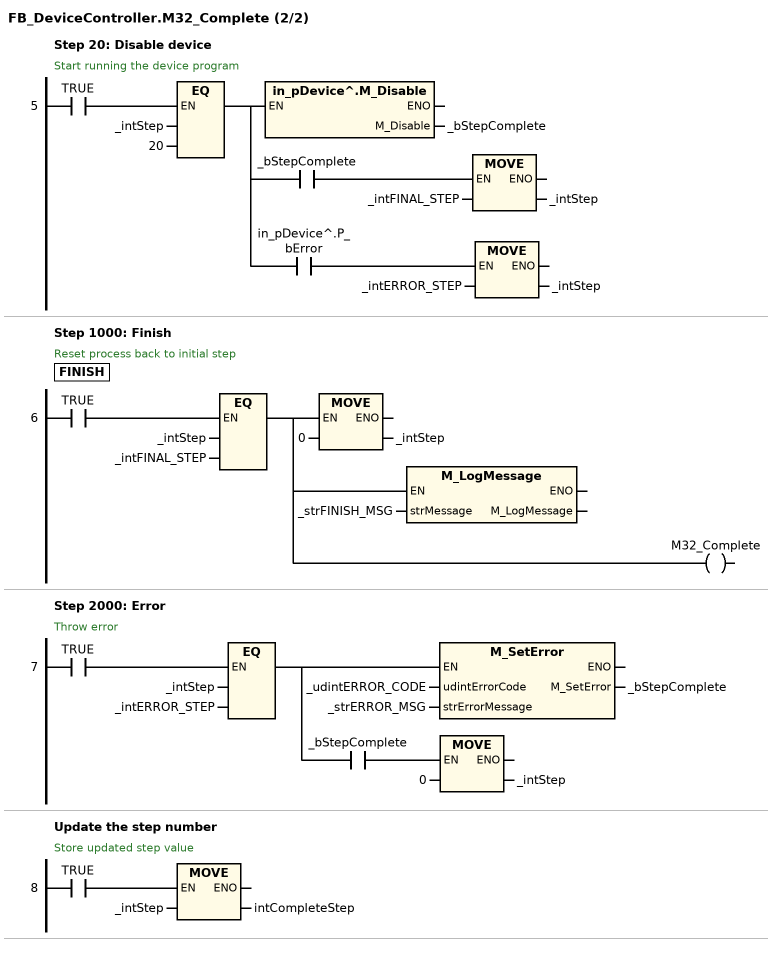
// NETWORK 5: Step 20: Disable device
// Start running the device program
_w6 := _intStep = 20;
IF _w6 THEN _bStepComplete := in_pDevice^.M_Disable(); END_IF
IF _w6 AND _bStepComplete THEN _intStep := _intFINAL_STEP; END_IF
IF _w6 AND in_pDevice^.P_bError THEN _intStep := _intERROR_STEP; END_IF

// NETWORK 6: Step 1000: Finish
// Reset process back to initial step
FINISH:
_w7 := _intStep = _intFINAL_STEP;
IF _w7 THEN _intStep := 0; END_IF
IF _w7 THEN M_LogMessage(strMessage := _strFINISH_MSG); END_IF
M32_Complete := _w7;

// NETWORK 7: Step 2000: Error
// Throw error
_w8 := _intStep = _intERROR_STEP;
IF _w8 THEN
    _bStepComplete := M_SetError(udintErrorCode := _udintERROR_CODE, strErrorMessage := _strERROR_MSG);
END_IF
IF _w8 AND _bStepComplete THEN _intStep := 0; END_IF

// NETWORK 8: Update the step number
// Store updated step value
intCompleteStep := _intStep;
END_METHOD

(* Pauses the device then returns TRUE. *)
METHOD M40_Hold : BOOL
VAR CONSTANT
	_udintERROR_CODE: UDINT := E_DeviceControllerError.HoldError;
	_strERROR_MSG: T_MaxString := 'Error while trying to hold device!';
	_intFINAL_STEP : INT := 1000;
	_intERROR_STEP : INT := 2000;
	_strSTART_MSG: T_MaxString := 'Holding device';
	_strFINISH_MSG: T_MaxString := 'Device held';
END_VAR
VAR
	_bStepComplete: BOOL;
	_intStep: INT;
END_VAR
VAR_INST // added by the converter: edge detectors and wires of the graphical bodies
    _w1, _w2, _w3, _w4, _w5, _w6, _w7 : BOOL;
END_VAR
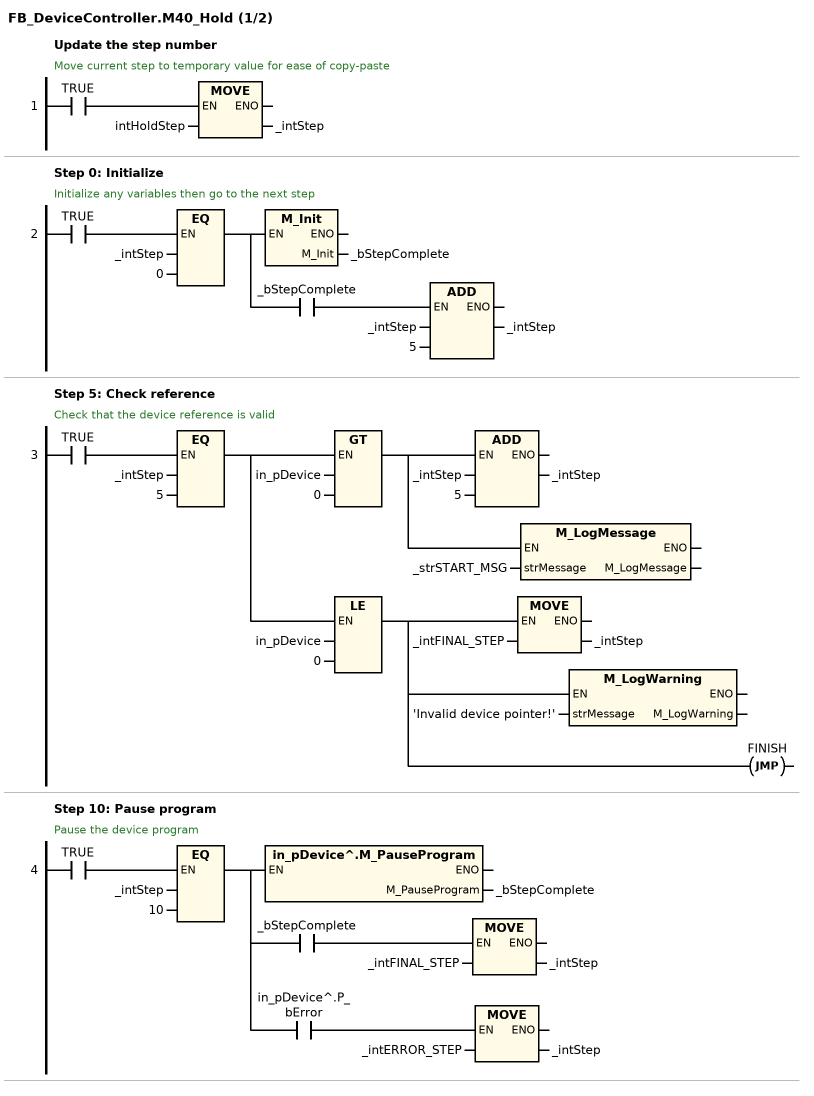
// NETWORK 1: Update the step number
// Move current step to temporary value for ease of copy-paste
_intStep := intHoldStep;

// NETWORK 2: Step 0: Initialize
// Initialize any variables then go to the next step
_w1 := _intStep = 0;
IF _w1 THEN _bStepComplete := M_Init(); END_IF
IF _w1 AND _bStepComplete THEN _intStep := _intStep + 5; END_IF

// NETWORK 3: Step 5: Check reference
// Check that the device reference is valid
_w2 := _intStep = 5;
_w3 := _w2 AND in_pDevice > 0;
IF _w3 THEN _intStep := _intStep + 5; END_IF
IF _w3 THEN M_LogMessage(strMessage := _strSTART_MSG); END_IF
_w4 := _w2 AND in_pDevice <= 0;
IF _w4 THEN _intStep := _intFINAL_STEP; END_IF
IF _w4 THEN M_LogWarning(strMessage := 'Invalid device pointer!'); END_IF
IF _w4 THEN JMP FINISH; END_IF

// NETWORK 4: Step 10: Pause program
// Pause the device program
_w5 := _intStep = 10;
IF _w5 THEN _bStepComplete := in_pDevice^.M_PauseProgram(); END_IF
IF _w5 AND _bStepComplete THEN _intStep := _intFINAL_STEP; END_IF
IF _w5 AND in_pDevice^.P_bError THEN _intStep := _intERROR_STEP; END_IF

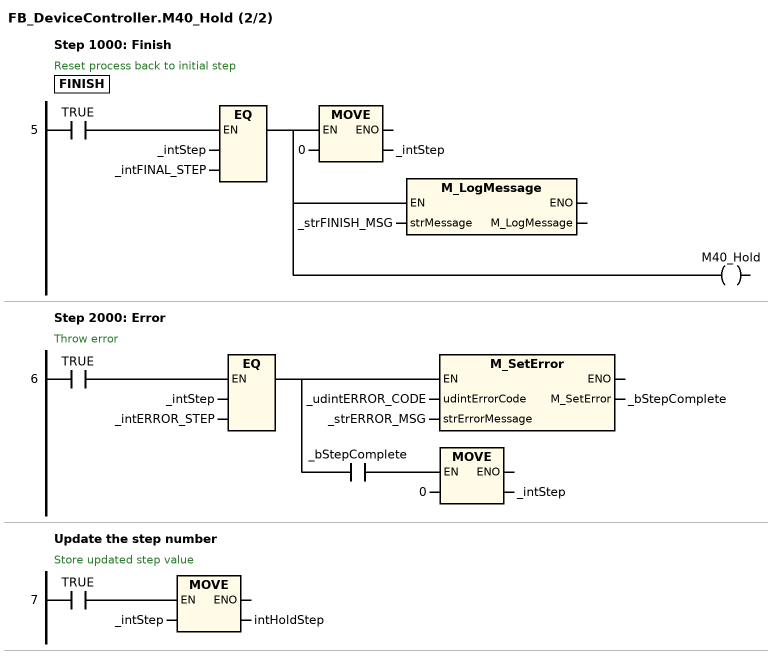
// NETWORK 5: Step 1000: Finish
// Reset process back to initial step
FINISH:
_w6 := _intStep = _intFINAL_STEP;
IF _w6 THEN _intStep := 0; END_IF
IF _w6 THEN M_LogMessage(strMessage := _strFINISH_MSG); END_IF
M40_Hold := _w6;

// NETWORK 6: Step 2000: Error
// Throw error
_w7 := _intStep = _intERROR_STEP;
IF _w7 THEN
    _bStepComplete := M_SetError(udintErrorCode := _udintERROR_CODE, strErrorMessage := _strERROR_MSG);
END_IF
IF _w7 AND _bStepComplete THEN _intStep := 0; END_IF

// NETWORK 7: Update the step number
// Store updated step value
intHoldStep := _intStep;
END_METHOD

(* Unpauses the device then returns TRUE. *)
METHOD M42_Unhold : BOOL
VAR CONSTANT
	_udintERROR_CODE: UDINT := E_DeviceControllerError.UnholdError;
	_strERROR_MSG: T_MaxString := 'Error while trying to unhold device!';
	_intFINAL_STEP : INT := 1000;
	_intERROR_STEP : INT := 2000;
	_strSTART_MSG: T_MaxString := 'Unholding device';
	_strFINISH_MSG: T_MaxString := 'Device unheld';
END_VAR
VAR
	_bStepComplete: BOOL;
	_intStep: INT;
END_VAR
VAR_INST // added by the converter: edge detectors and wires of the graphical bodies
    _w1, _w2, _w3, _w4, _w5, _w6, _w7 : BOOL;
END_VAR
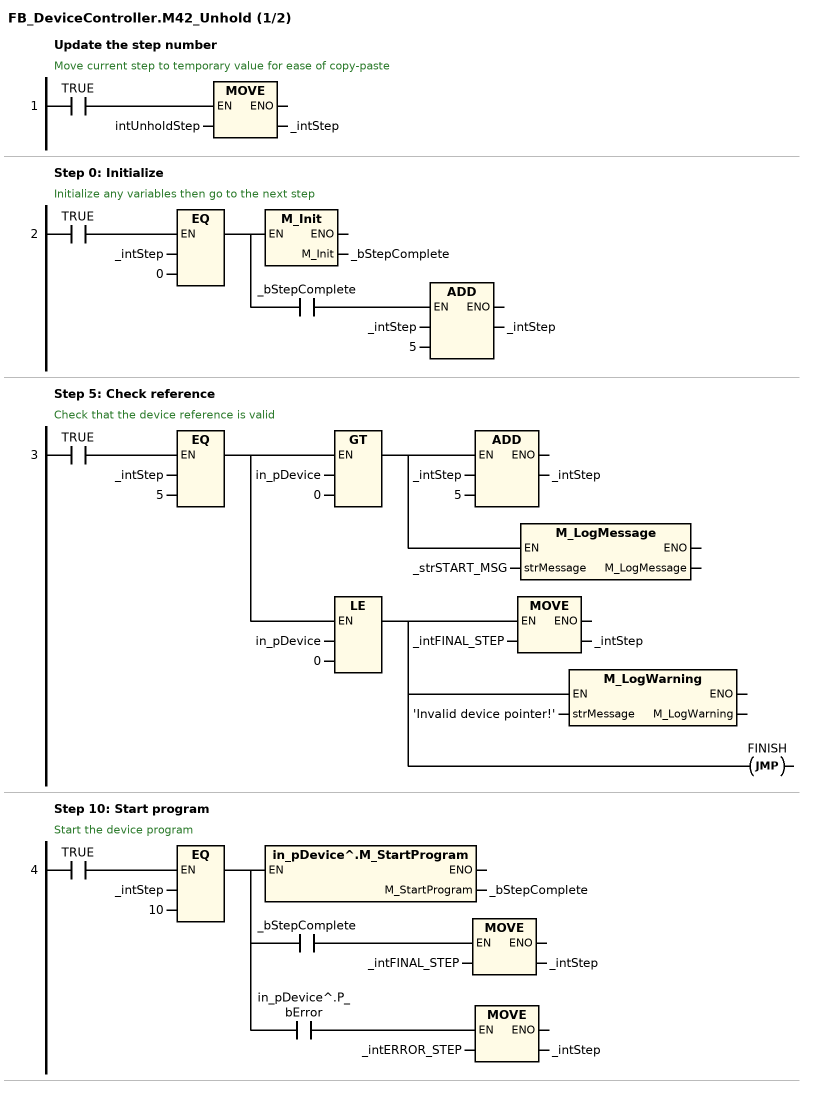
// NETWORK 1: Update the step number
// Move current step to temporary value for ease of copy-paste
_intStep := intUnholdStep;

// NETWORK 2: Step 0: Initialize
// Initialize any variables then go to the next step
_w1 := _intStep = 0;
IF _w1 THEN _bStepComplete := M_Init(); END_IF
IF _w1 AND _bStepComplete THEN _intStep := _intStep + 5; END_IF

// NETWORK 3: Step 5: Check reference
// Check that the device reference is valid
_w2 := _intStep = 5;
_w3 := _w2 AND in_pDevice > 0;
IF _w3 THEN _intStep := _intStep + 5; END_IF
IF _w3 THEN M_LogMessage(strMessage := _strSTART_MSG); END_IF
_w4 := _w2 AND in_pDevice <= 0;
IF _w4 THEN _intStep := _intFINAL_STEP; END_IF
IF _w4 THEN M_LogWarning(strMessage := 'Invalid device pointer!'); END_IF
IF _w4 THEN JMP FINISH; END_IF

// NETWORK 4: Step 10: Start program
// Start the device program
_w5 := _intStep = 10;
IF _w5 THEN _bStepComplete := in_pDevice^.M_StartProgram(); END_IF
IF _w5 AND _bStepComplete THEN _intStep := _intFINAL_STEP; END_IF
IF _w5 AND in_pDevice^.P_bError THEN _intStep := _intERROR_STEP; END_IF

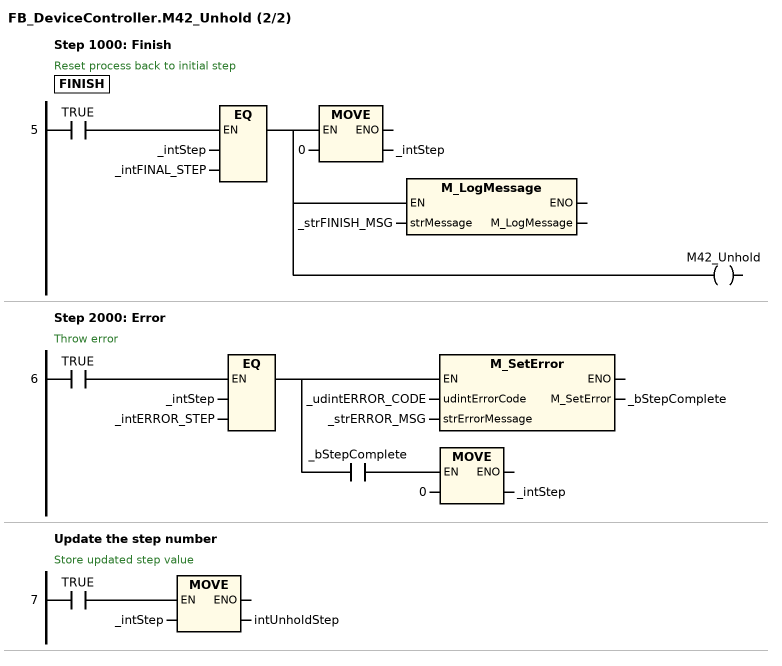
// NETWORK 5: Step 1000: Finish
// Reset process back to initial step
FINISH:
_w6 := _intStep = _intFINAL_STEP;
IF _w6 THEN _intStep := 0; END_IF
IF _w6 THEN M_LogMessage(strMessage := _strFINISH_MSG); END_IF
M42_Unhold := _w6;

// NETWORK 6: Step 2000: Error
// Throw error
_w7 := _intStep = _intERROR_STEP;
IF _w7 THEN
    _bStepComplete := M_SetError(udintErrorCode := _udintERROR_CODE, strErrorMessage := _strERROR_MSG);
END_IF
IF _w7 AND _bStepComplete THEN _intStep := 0; END_IF

// NETWORK 7: Update the step number
// Store updated step value
intUnholdStep := _intStep;
END_METHOD

(* Pauses the device then returns TRUE. *)
METHOD M50_Suspend : BOOL
VAR CONSTANT
	_udintERROR_CODE: UDINT := E_DeviceControllerError.SuspendError;
	_strERROR_MSG: T_MaxString := 'Error while trying to suspend device!';
	_intFINAL_STEP : INT := 1000;
	_intERROR_STEP : INT := 2000;
	_strSTART_MSG: T_MaxString := 'Suspending device';
	_strFINISH_MSG: T_MaxString := 'Device suspended';
END_VAR
VAR
	_bStepComplete: BOOL;
	_intStep: INT;
END_VAR
VAR_INST // added by the converter: edge detectors and wires of the graphical bodies
    _w1, _w2, _w3, _w4, _w5, _w6, _w7 : BOOL;
END_VAR
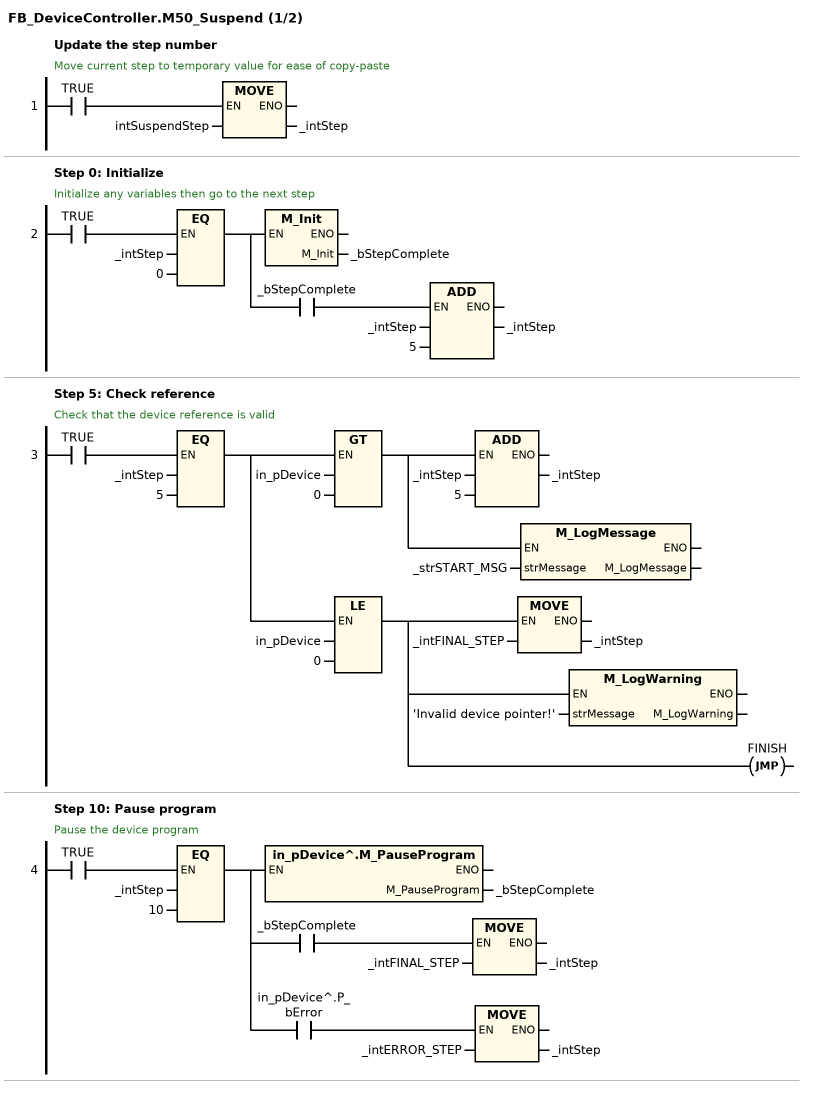
// NETWORK 1: Update the step number
// Move current step to temporary value for ease of copy-paste
_intStep := intSuspendStep;

// NETWORK 2: Step 0: Initialize
// Initialize any variables then go to the next step
_w1 := _intStep = 0;
IF _w1 THEN _bStepComplete := M_Init(); END_IF
IF _w1 AND _bStepComplete THEN _intStep := _intStep + 5; END_IF

// NETWORK 3: Step 5: Check reference
// Check that the device reference is valid
_w2 := _intStep = 5;
_w3 := _w2 AND in_pDevice > 0;
IF _w3 THEN _intStep := _intStep + 5; END_IF
IF _w3 THEN M_LogMessage(strMessage := _strSTART_MSG); END_IF
_w4 := _w2 AND in_pDevice <= 0;
IF _w4 THEN _intStep := _intFINAL_STEP; END_IF
IF _w4 THEN M_LogWarning(strMessage := 'Invalid device pointer!'); END_IF
IF _w4 THEN JMP FINISH; END_IF

// NETWORK 4: Step 10: Pause program
// Pause the device program
_w5 := _intStep = 10;
IF _w5 THEN _bStepComplete := in_pDevice^.M_PauseProgram(); END_IF
IF _w5 AND _bStepComplete THEN _intStep := _intFINAL_STEP; END_IF
IF _w5 AND in_pDevice^.P_bError THEN _intStep := _intERROR_STEP; END_IF

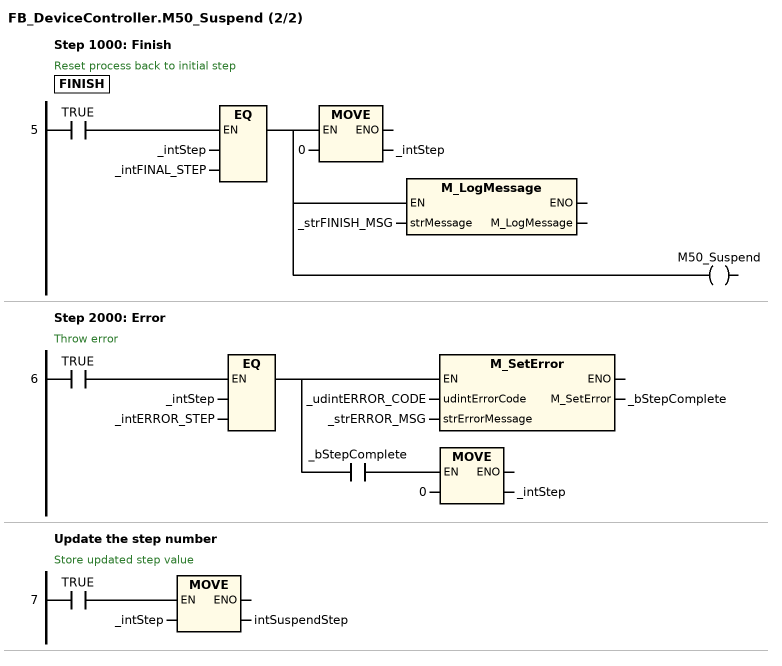
// NETWORK 5: Step 1000: Finish
// Reset process back to initial step
FINISH:
_w6 := _intStep = _intFINAL_STEP;
IF _w6 THEN _intStep := 0; END_IF
IF _w6 THEN M_LogMessage(strMessage := _strFINISH_MSG); END_IF
M50_Suspend := _w6;

// NETWORK 6: Step 2000: Error
// Throw error
_w7 := _intStep = _intERROR_STEP;
IF _w7 THEN
    _bStepComplete := M_SetError(udintErrorCode := _udintERROR_CODE, strErrorMessage := _strERROR_MSG);
END_IF
IF _w7 AND _bStepComplete THEN _intStep := 0; END_IF

// NETWORK 7: Update the step number
// Store updated step value
intSuspendStep := _intStep;
END_METHOD

(* Unpauses the device then returns TRUE. *)
METHOD M52_Unsuspend : BOOL
VAR CONSTANT
	_udintERROR_CODE: UDINT := E_DeviceControllerError.ResetError;
	_strERROR_MSG: T_MaxString := 'Error while trying to reset device!';
	_intFINAL_STEP : INT := 1000;
	_intERROR_STEP : INT := 2000;
	_strSTART_MSG: T_MaxString := 'Unsuspending device';
	_strFINISH_MSG: T_MaxString := 'Device unsuspended';
END_VAR
VAR
	_bStepComplete: BOOL;
	_intStep: INT;
END_VAR
VAR_INST // added by the converter: edge detectors and wires of the graphical bodies
    _w1, _w2, _w3, _w4, _w5, _w6, _w7 : BOOL;
END_VAR
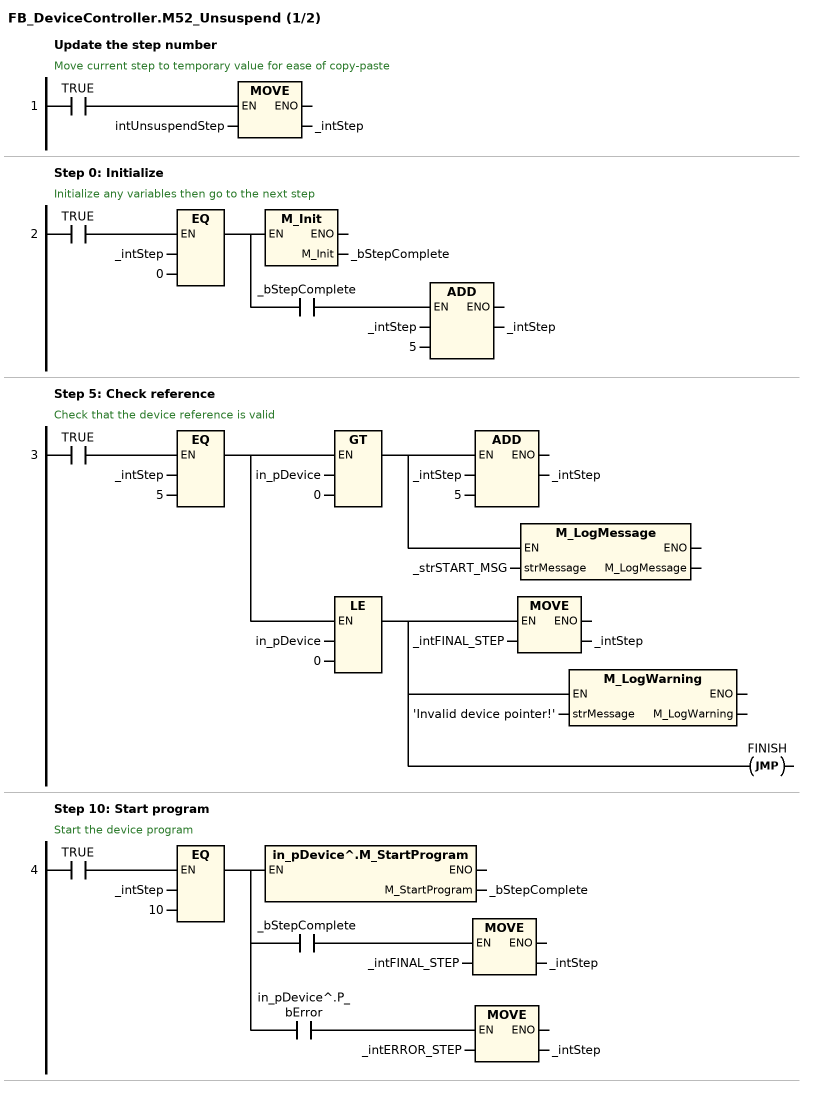
// NETWORK 1: Update the step number
// Move current step to temporary value for ease of copy-paste
_intStep := intUnsuspendStep;

// NETWORK 2: Step 0: Initialize
// Initialize any variables then go to the next step
_w1 := _intStep = 0;
IF _w1 THEN _bStepComplete := M_Init(); END_IF
IF _w1 AND _bStepComplete THEN _intStep := _intStep + 5; END_IF

// NETWORK 3: Step 5: Check reference
// Check that the device reference is valid
_w2 := _intStep = 5;
_w3 := _w2 AND in_pDevice > 0;
IF _w3 THEN _intStep := _intStep + 5; END_IF
IF _w3 THEN M_LogMessage(strMessage := _strSTART_MSG); END_IF
_w4 := _w2 AND in_pDevice <= 0;
IF _w4 THEN _intStep := _intFINAL_STEP; END_IF
IF _w4 THEN M_LogWarning(strMessage := 'Invalid device pointer!'); END_IF
IF _w4 THEN JMP FINISH; END_IF

// NETWORK 4: Step 10: Start program
// Start the device program
_w5 := _intStep = 10;
IF _w5 THEN _bStepComplete := in_pDevice^.M_StartProgram(); END_IF
IF _w5 AND _bStepComplete THEN _intStep := _intFINAL_STEP; END_IF
IF _w5 AND in_pDevice^.P_bError THEN _intStep := _intERROR_STEP; END_IF

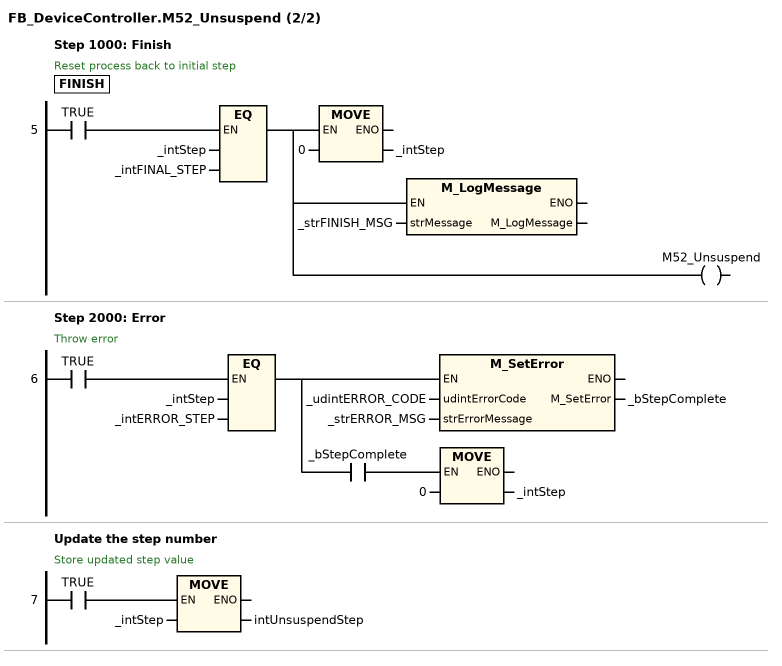
// NETWORK 5: Step 1000: Finish
// Reset process back to initial step
FINISH:
_w6 := _intStep = _intFINAL_STEP;
IF _w6 THEN _intStep := 0; END_IF
IF _w6 THEN M_LogMessage(strMessage := _strFINISH_MSG); END_IF
M52_Unsuspend := _w6;

// NETWORK 6: Step 2000: Error
// Throw error
_w7 := _intStep = _intERROR_STEP;
IF _w7 THEN
    _bStepComplete := M_SetError(udintErrorCode := _udintERROR_CODE, strErrorMessage := _strERROR_MSG);
END_IF
IF _w7 AND _bStepComplete THEN _intStep := 0; END_IF

// NETWORK 7: Update the step number
// Store updated step value
intUnsuspendStep := _intStep;
END_METHOD

END_FUNCTION_BLOCK

// Concrete/Obsolete/FB_DeviceTestStation_Old
{attribute 'obsolete' := 'Use FB_DeviceTestStation'} 
FUNCTION_BLOCK FB_DeviceTestStation_Old EXTENDS FB_Station IMPLEMENTS I_Stateful
VAR_INPUT
	ref_fbDevice: REFERENCE TO FB_Device; // The device to be tested
	
	in_bAbortBtn: BOOL; // Abort from any abortable states
	in_bClearBtn: BOOL; // Clear the abort state and any errors
	in_bStopBtn: BOOL; // Stop from any stoppable states
	in_bResetBtn: BOOL; // Return to the idle state from stopped or completed
	in_bStartBtn: BOOL; // Start from idle or restart from held or suspended
	in_bCompleteBtn: BOOL; // Exit the execute step to the complete step
	in_bHoldBtn: BOOL; // Hold the machine while in execute state
	in_bSuspendBtn: BOOL; // Suspend the machine while in execute state
	
	in_strProgram: T_MaxString; // Program to load when testing program loading
END_VAR
VAR_OUTPUT
	out_bAbortTested: BOOL; // Gets set to TRUE once M_Abort on ref_fbDevice has been tested once
	
	out_bConnectTested: BOOL;  // Gets set to TRUE once M_Connect on ref_fbDevice has been tested once
	out_bDisconnectTested: BOOL;  // Gets set to TRUE once M_Disconnect on ref_fbDevice has been tested once
	
	out_bEnableTested: BOOL; // Gets set to TRUE once M_Enable on ref_fbDevice has been tested once
	out_bDisableTested: BOOL; // Gets set to TRUE once M_Disable on ref_fbDevice has been tested once
	
	out_bPowerOnTested: BOOL; // Gets set to TRUE once M_PowerOn on ref_fbDevice has been tested once
	out_bPowerOffTested: BOOL; // Gets set to TRUE once M_PowerOff on ref_fbDevice has been tested once
	
	out_bLoadProgramTested: BOOL; // Gets set to TRUE once M_LoadProgram on ref_fbDevice has been tested once
	out_bStartProgramTested: BOOL; // Gets set to TRUE once M_StartProgram on ref_fbDevice has been tested once
	out_bStopProgramTested: BOOL; // Gets set to TRUE once M_StopProgram on ref_fbDevice has been tested once
	out_bPauseProgramTested: BOOL; // Gets set to TRUE once M_PauseProgram on ref_fbDevice has been tested once
	out_bUnpauseProgramTested: BOOL; // Gets set to TRUE once M_StartProgram on ref_fbDevice has been tested once after M_PauseProgram was used
	out_bStopPausedProgramTested: BOOL; // Gets set to TRUE once M_StopProgram on ref_fbDevice has been tested once after M_PauseProgram was used
	
	out_bResetTested: BOOL; // Gets set to TRUE once M_Reset on ref_fbDevice has been tested once
END_VAR
VAR
	bDeviceReset: BOOL;
	
	bDeviceConnected: BOOL;
	bDeviceDisconnected: BOOL;
	
	bDevicePoweredOn: BOOL;
	bDevicePoweredOff: BOOL;
	
	bDeviceEnabled: BOOL;
	bDeviceDisabled: BOOL;
	
	bDeviceProgramLoaded: BOOL;
	bDeviceProgramStarted: BOOL;
	bDeviceProgramStopped: BOOL;
	bDeviceProgramPaused: BOOL;

	// Device test trackers
	fbDeviceAborted: R_TRIG;
	fbDeviceReset: F_TRIG;
	fbDeviceConnected: R_TRIG;
	fbDeviceDisconnected: F_TRIG;
	fbDeviceEnabled: R_TRIG;
	fbDeviceDisabled: F_TRIG;
	fbDevicePoweredOn: R_TRIG;
	fbDevicePoweredOff: F_TRIG;
	fbDeviceProgramLoaded: R_TRIG;
	enumLastState: E_ProgramState;
END_VAR

THIS^.M_SetDevice(1, ref_fbDevice);

A_StateMachine();

A_DeviceTestTracking();

(* Runs for a single cycle when entering the aborting state. *)
METHOD M000_Aborting_Entry : BOOL
THIS^.M_LogMessage('Aborting');
END_METHOD

(* The 'Aborting' state can be entered at any time while within the 'abortable'
section of the state machine. It is typically entered in response to an 'Abort'
command or a critical fault. The logic should safely but rapidly bring the
components of the module to a stop while maintaining as much information about
the pre-abort scenario as possible. *)
METHOD M001_Aborting : BOOL
VAR_OUTPUT
	(* This should be set to true once all components of the module have safely
	come to a stop. Once set to true, the state machine will move to the
	'Aborted' state. *)
	bAborted	: BOOL;
END_VAR
// Go to the aborted state once the device is aborted
bAborted := ref_fbDevice.M_Abort();
END_METHOD

(* Runs for a single cycle when exiting the aborting state. *)
METHOD M002_Aborting_Exit : BOOL
END_METHOD

(* Runs for a single cycle when entering the aborted state. *)
METHOD M010_Aborted_Entry : BOOL
THIS^.M_LogMessage('Aborted');
END_METHOD

(* This state is entered after the aborting state completes, and should
not modify anything in the module while awaiting an explicit 'Clear' command. *)
METHOD M011_Aborted : BOOL
VAR_OUTPUT
	(* This should be set to true once an explicit 'Clear' command is received.
	Once set to true, the state machine will move to the 'Clearing' state. *)
	bClear	: BOOL;
END_VAR
// Only go to clearing state if clear button is pressed
bClear := in_bClearBtn;
END_METHOD

(* Runs for a single cycle when exiting the aborted state. *)
METHOD M012_Aborted_Exit : BOOL
END_METHOD

(* Runs for a single cycle when entering the clearing state. *)
METHOD M020_Clearing_Entry : BOOL
THIS^.M_LogMessage('Clearing');
END_METHOD

(* This state should clear any faults and reset any safety features related
to the module, as well as perform actions similar to the 'Stopping' state
if they were not already performed while aborting. *)
METHOD M021_Clearing : BOOL
VAR_OUTPUT
	(* This should be set to true once the safety state of all module
	components are reset and all errors are cleared. *)
	bCleared	: BOOL;
	(* This should be set to true if a potentially hazardous error or a safety
	fault has occurred in any tasks. Once set to true, the state machine will
	move to the 'Aborting' state. *)
	bAbort	: BOOL;
END_VAR
// Exit once the device is reset
bCleared := ref_fbDevice.M_Reset();

// If device is reset, clear module errors
IF bCleared THEN
	THIS^.M_ClearError();
END_IF

// If the device has an error, abort
IF ref_fbDevice.P_bError THEN
	THIS^.M_SetError(200, 'Error on fbDevice!');
	bAbort := TRUE;
	
// Abort if abort button is pressed
ELSIF in_bAbortBtn THEN
	THIS^.M_SetError(100, 'Abort button pressed!');
	bAbort := TRUE;
END_IF
END_METHOD

(* Runs for a single cycle when exiting the clearing state. *)
METHOD M022_Clearing_Exit : BOOL
END_METHOD

(* Runs for a single cycle when entering the stopping state. *)
METHOD M100_Stopping_Entry : BOOL
THIS^.M_LogMessage('Stopping');

// Reset device status variables
bDeviceProgramStopped := FALSE;
bDeviceDisabled := FALSE;
bDevicePoweredOff := FALSE;
END_METHOD

(* This state can be entered from anywhere within the 'stoppable' group of
states. This state should safely bring the components of the module to a
controlled stop and then move to the 'Stopped' state once completed. *)
METHOD M101_Stopping : BOOL
VAR_OUTPUT
	(* This should be set to true once all relevant components have come to a
	controlled stop. Once set to true, the state machine will move to the
	'Stopped' state. *)
	bStopped	: BOOL;
	(* This should be set to true if a potentially hazardous error or a safety
	fault has occurred in any tasks. Once set to true, the state machine will
	move to the 'Aborting' state. *)
	bAbort	: BOOL;
END_VAR
// If the device is connected, stop and disable it
IF ref_fbDevice.P_bConnected THEN
	
	// Stop the program
	IF NOT bDeviceProgramStopped THEN
		bDeviceProgramStopped := ref_fbDevice.M_StopProgram();
		
	// Disable the device
	ELSIF NOT bDeviceDisabled THEN
		bDeviceDisabled := ref_fbDevice.M_Disable();
	
	// Power off the device
	ELSIF NOT bDevicePoweredOff THEN
		bDevicePoweredOff := ref_fbDevice.M_PowerOff();
		
	// Exit once stopped and disabled
	ELSE
		bStopped := TRUE;
	END_IF
	
// If the device is not connected, it can be considered to be stopped
ELSE
	bStopped := TRUE;
END_IF

// If the device has an error, abort
IF ref_fbDevice.P_bError THEN
	THIS^.M_SetError(200, 'Error on fbDevice!');
	bAbort := TRUE;
	
// Abort if abort button is pressed
ELSIF in_bAbortBtn THEN
	THIS^.M_SetError(100, 'Abort button pressed!');
	bAbort := TRUE;
END_IF
END_METHOD

(* Runs for a single cycle when exiting the stopping state. *)
METHOD M102_Stopping_Exit : BOOL
END_METHOD

(* Runs for a single cycle when entering the stopped state. *)
METHOD M110_Stopped_Entry : BOOL
THIS^.M_LogMessage('Stopped');
END_METHOD

(* The machine should be stationary and awaiting an explicit 'Reset' command
while in this state. Once the 'Reset' command is received, the state machine
will move to the 'Resetting' state. *)
METHOD M111_Stopped : BOOL
VAR_OUTPUT
	(* This should be set to true if an explicit reset command is received.
	Once set to true, the state machine will move to the 'Resetting' state. *)
	bReset	: BOOL;
	(* This should be set to true if a potentially hazardous error or a safety
	fault has occurred in any tasks. Once set to true, the state machine will
	move to the 'Aborting' state. *)
	bAbort	: BOOL;
END_VAR
// Go to the resetting state if the reset button is pressed
bReset := in_bResetBtn;

// If the device has an error, abort
IF ref_fbDevice.P_bError THEN
	THIS^.M_SetError(200, 'Error on fbDevice!');
	bAbort := TRUE;
	
// Abort if abort button is pressed
ELSIF in_bAbortBtn THEN
	THIS^.M_SetError(100, 'Abort button pressed!');
	bAbort := TRUE;
END_IF
END_METHOD

(* Runs for a single cycle when exiting the stopped state. *)
METHOD M112_Stopped_Exit : BOOL
END_METHOD

(* Runs for a single cycle when entering the resetting state. *)
METHOD M200_Resetting_Entry : BOOL
THIS^.M_LogMessage('Resetting');

// Reset device status variables
bDeviceDisconnected := FALSE;
bDeviceConnected := FALSE;
bDeviceReset := FALSE;
END_METHOD

(* This state should place the module and all of its components into a safe
energized idle state where it will wait for a start command. Once all tasks are
complete, it will move to the 'Idle' state. No external movement should occur
as a result of this state. *)
METHOD M201_Resetting : BOOL
VAR_OUTPUT
	(* Set this to true once the module is energized and ready to start.
	Once set to true, the state machine will move to the 'Idle' state. *)
	bIdle	: BOOL;
	(* This should be set to true if an external source requests that the module
	exit its current state and come to a controlled stop. Once set to true, the
	state machine will move to the 'Stopping' state. *)
	bStop	: BOOL;
	(* This should be set to true if a potentially hazardous error or a safety
	fault has occurred in any tasks. Once set to true, the state machine will
	move to the 'Aborting' state. *)
	bAbort	: BOOL;
END_VAR
// Stop if stop button is pressed
bStop := in_bStopBtn;

// Disconnect the device to reset the connection
IF NOT bDeviceDisconnected THEN
	bDeviceDisconnected := ref_fbDevice.M_Disconnect();
	
// Connect (or reconnect) the device
ELSIF NOT bDeviceConnected THEN
	bDeviceConnected := ref_fbDevice.M_Connect();
	
// Reset the device
ELSIF NOT bDeviceReset THEN
	bDeviceReset := ref_fbDevice.M_Reset();

// Once reconnected and reset, go to the idle state
ELSE
	bIdle := TRUE;
END_IF

// If the device has an error, abort
IF ref_fbDevice.P_bError THEN
	THIS^.M_SetError(200, 'Error on fbDevice!');
	bAbort := TRUE;
	
// Abort if abort button is pressed
ELSIF in_bAbortBtn THEN
	THIS^.M_SetError(100, 'Abort button pressed!');
	bAbort := TRUE;

END_IF
END_METHOD

(* Runs for a single cycle when exiting the resetting state. *)
METHOD M202_Resetting_Exit : BOOL
END_METHOD

(* Runs for a single cycle when entering the idle state. *)
METHOD M210_Idle_Entry : BOOL
THIS^.M_LogMessage('Idle');
END_METHOD

(* This state should maintain the status of the module and its components that
was set by the resetting step while awaiting an explicit 'Start' command. *)
METHOD M211_Idle : BOOL
VAR_OUTPUT
	(* This should be set to true if an explicit 'Start' command is received.
	Once set to true, the state machine will move to the 'Starting' state. *)
	bStart	: BOOL;
	(* This should be set to true if an external source requests that the module
	exit its current state and come to a controlled stop. Once set to true, the
	state machine will move to the 'Stopping' state. *)
	bStop	: BOOL;
	(* This should be set to true if a potentially hazardous error or a safety
	fault has occurred in any tasks. Once set to true, the state machine will
	move to the 'Aborting' state. *)
	bAbort	: BOOL;
END_VAR
// Start if start button is pressed
bStart := in_bStartBtn;

// Stop if stop button is pressed
bStop := in_bStopBtn;

// If the device has an error, abort
IF ref_fbDevice.P_bError THEN
	THIS^.M_SetError(200, 'Error on fbDevice!');
	bAbort := TRUE;
	
// Abort if abort button is pressed
ELSIF in_bAbortBtn THEN
	THIS^.M_SetError(100, 'Abort button pressed!');
	bAbort := TRUE;

END_IF
END_METHOD

(* Runs for a single cycle when exiting the idle state. *)
METHOD M212_Idle_Exit : BOOL
END_METHOD

(* Runs for a single cycle when entering the starting state. *)
METHOD M300_Starting_Entry : BOOL
THIS^.M_LogMessage('Starting');

// Reset device status variables
bDeviceProgramLoaded := FALSE;
bDevicePoweredOn := FALSE;
bDeviceEnabled := FALSE;
bDeviceProgramStarted := FALSE;
END_METHOD

(* This state should make any final preparations needed for the 'Execute' state
prior to entering the 'Execute' state. *)
METHOD M301_Starting : BOOL
VAR_OUTPUT
	(* This should be set to true once the module and its components are fully
	prepared for process execution. Once set to true, the state machine will
	move to the 'Execute' state. *)
	bStarted	: BOOL;
	(* This should be set to true if an external source requests that the module
	exit its current state and come to a controlled stop. Once set to true, the
	state machine will move to the 'Stopping' state. *)
	bStop	: BOOL;
	(* This should be set to true if a potentially hazardous error or a safety
	fault has occurred in any tasks. Once set to true, the state machine will
	move to the 'Aborting' state. *)
	bAbort	: BOOL;
END_VAR
// Stop if stop button is pressed
bStop := in_bStopBtn;

// Load a program on the device
IF NOT bDeviceProgramLoaded THEN
	bDeviceProgramLoaded := ref_fbDevice.M_LoadProgram(in_strProgram);

// Power on the device
ELSIF NOT bDevicePoweredOn THEN
	bDevicePoweredOn := ref_fbDevice.M_PowerOn();

// Enable the device
ELSIF NOT bDeviceEnabled THEN
	bDeviceEnabled := ref_fbDevice.M_Enable();
	
// Start the device program
ELSIF NOT bDeviceProgramStarted THEN
	bDeviceProgramStarted := ref_fbDevice.M_StartProgram();

// Go to execute state once device program is started
ELSE
	bStarted := TRUE;
END_IF

// If the device has an error, abort
IF ref_fbDevice.P_bError THEN
	THIS^.M_SetError(200, 'Error on fbDevice!');
	bAbort := TRUE;
	
// Abort if abort button is pressed
ELSIF in_bAbortBtn THEN
	THIS^.M_SetError(100, 'Abort button pressed!');
	bAbort := TRUE;

END_IF
END_METHOD

(* Runs for a single cycle when exiting the starting state. *)
METHOD M302_Starting_Exit : BOOL
END_METHOD

(* Runs for a single cycle when entering the execute state. *)
METHOD M310_Execute_Entry : BOOL
THIS^.M_LogMessage('Execute');
END_METHOD

(* The module should remain in this state while it is actively performing
automated tasks. Once all work is finished the state machine should move to the
'Completing' state. *)
METHOD M311_Execute : BOOL
VAR_OUTPUT
	(* This should be set to true once all tasks are complete and automated
	execution should be ended. Once set to true, the state machine will move to
	the 'Completing' state. *)
	bFinished	: BOOL;
	(* This should be set to true as a result of an explicit 'Hold' command
	or if internal conditions require the module to stop operation without
	completely exiting the execution sequence. Once set to true, the state
	machine will move to the 'Holding' state. *)
	bHold	: BOOL;
	(* This should be set to true if external conditions require the module to
	suspend operation until the external conditions are cleared. Once set to
	true, the state machine will move to the 'Suspending' state. *)
	bSuspend	: BOOL;
	(* This should be set to true if an external source requests that the module
	exit its current state and come to a controlled stop. Once set to true, the
	state machine will move to the 'Stopping' state. *)
	bStop	: BOOL;
	(* This should be set to true if a potentially hazardous error or a safety
	fault has occurred in any tasks. Once set to true, the state machine will
	move to the 'Aborting' state. *)
	bAbort	: BOOL;
END_VAR
// Complete if the complete button is pressed
bFinished := in_bCompleteBtn;

// Hold if the hold button is pressed
bHold := in_bHoldBtn;

// Suspend if the suspend button is pressed
bSuspend := in_bSuspendBtn;

// Stop if the stop button is pressed
bStop := in_bStopBtn;

// If the device has an error, abort
IF ref_fbDevice.P_bError THEN
	THIS^.M_SetError(200, 'Error on fbDevice!');
	bAbort := TRUE;
	
// Abort if abort button is pressed
ELSIF in_bAbortBtn THEN
	THIS^.M_SetError(100, 'Abort button pressed!');
	bAbort := TRUE;
END_IF
END_METHOD

(* Runs for a single cycle when exiting the execute state. *)
METHOD M312_Execute_Exit : BOOL
END_METHOD

(* Runs for a single cycle when entering the completing state. *)
METHOD M320_Completing_Entry : BOOL
THIS^.M_LogMessage('Completing');

// Reset device status variables
bDeviceProgramStopped := FALSE;
bDeviceDisabled := FALSE;
END_METHOD

(* This state will perform any post-execution tasks prior to moving to the
'Completed' state. *)
METHOD M321_Completing : BOOL
VAR_OUTPUT
	(* Move to the Complete state*)
	bCompleted	: BOOL;
	(* This should be set to true if an external source requests that the module
	exit its current state and come to a controlled stop. Once set to true, the
	state machine will move to the 'Stopping' state. *)
	bStop	: BOOL;
	(* This should be set to true if a potentially hazardous error or a safety
	fault has occurred in any tasks. Once set to true, the state machine will
	move to the 'Aborting' state. *)
	bAbort	: BOOL;
END_VAR
// Stop the program on the device
IF NOT bDeviceProgramStopped THEN
	bDeviceProgramStopped := ref_fbDevice.M_StopProgram();
	
// Disable the device
ELSIF NOT bDeviceDisabled THEN
	bDeviceDisabled := ref_fbDevice.M_Disable();
	
// Once stoppe and disabled, execution is complete
ELSE
	bCompleted := TRUE;
END_IF

// Stop if the stop button is pressed
bStop := in_bStopBtn;

// If the device has an error, abort
IF ref_fbDevice.P_bError THEN
	THIS^.M_SetError(200, 'Error on fbDevice!');
	bAbort := TRUE;
	
// Abort if abort button is pressed
ELSIF in_bAbortBtn THEN
	THIS^.M_SetError(100, 'Abort button pressed!');
	bAbort := TRUE;
END_IF
END_METHOD

(* Runs for a single cycle when exiting the completing state. *)
METHOD M322_Completing_Exit : BOOL
END_METHOD

(* Runs for a single cycle when entering the complete state. *)
METHOD M330_Complete_Entry : BOOL
THIS^.M_LogMessage('Complete');
END_METHOD

(* The module should remain stationary within this state while maintaing any
execution statistics and awaiting an explicit 'Return' command. *)
METHOD M331_Complete : BOOL
VAR_OUTPUT
	(* This should be set to true if an explicit 'Return' command is received.
	Once set to true, the state machine will move to the 'Resetting' state. *)
	bReturn	: BOOL;
	(* This should be set to true if an external source requests that the module
	exit its current state and come to a controlled stop. Once set to true, the
	state machine will move to the 'Stopping' state. *)
	bStop	: BOOL;
	(* This should be set to true if a potentially hazardous error or a safety
	fault has occurred in any tasks. Once set to true, the state machine will
	move to the 'Aborting' state. *)
	bAbort	: BOOL;
END_VAR
// Return if the reset button is pressed
bReturn := in_bResetBtn;

// Stop if the stop button is pressed
bStop := in_bStopBtn;

// If the device has an error, abort
IF ref_fbDevice.P_bError THEN
	THIS^.M_SetError(200, 'Error on fbDevice!');
	bAbort := TRUE;
	
// Abort if abort button is pressed
ELSIF in_bAbortBtn THEN
	THIS^.M_SetError(100, 'Abort button pressed!');
	bAbort := TRUE;
END_IF
END_METHOD

(* Runs for a single cycle when exiting the complete state. *)
METHOD M332_Complete_Exit : BOOL
END_METHOD

(* Runs for a single cycle when entering the holding state. *)
METHOD M400_Holding_Entry : BOOL
THIS^.M_LogMessage('Holding');

// Reset device state variables
bDeviceProgramPaused := FALSE;
END_METHOD

(* This state should safely pause task executions without completely ending or
resetting them. *)
METHOD M401_Holding : BOOL
VAR_OUTPUT
	(* This should be set to true once all execution tasks are safely paused.
	Once set to true, the state machine will move to the 'Held' state. *)
	bHeld	: BOOL;
	(* This should be set to true if an external source requests that the module
	exit its current state and come to a controlled stop. Once set to true, the
	state machine will move to the 'Stopping' state. *)
	bStop	: BOOL;
	(* This should be set to true if a potentially hazardous error or a safety
	fault has occurred in any tasks. Once set to true, the state machine will
	move to the 'Aborting' state. *)
	bAbort	: BOOL;
END_VAR
// Pause the device
IF NOT bDeviceProgramPaused THEN
	bDeviceProgramPaused := ref_fbDevice.M_PauseProgram();
	
// Once the device is paused, done holding
ELSE
	bHeld := TRUE;
END_IF

// Stop if the stop button is pressed
bStop := in_bStopBtn;

// If the device has an error, abort
IF ref_fbDevice.P_bError THEN
	THIS^.M_SetError(200, 'Error on fbDevice!');
	bAbort := TRUE;
	
// Abort if abort button is pressed
ELSIF in_bAbortBtn THEN
	THIS^.M_SetError(100, 'Abort button pressed!');
	bAbort := TRUE;
END_IF
END_METHOD

(* Runs for a single cycle when exiting the holding state. *)
METHOD M402_Holding_Exit : BOOL
END_METHOD

(* Runs for a single cycle when entering the held state. *)
METHOD M410_Held_Entry : BOOL
THIS^.M_LogMessage('Held');
END_METHOD

(* In this state the most recent execution status should be maintained while
awaiting an explicit 'Unhold' command once internal conditions are satisfactory. *)
METHOD M411_Held : BOOL
VAR_OUTPUT
	(* This should be set to true if an explicit 'Unhold' command is received.
	Once set to true, the state machine will move to the 'Unholding' state. *)
	bUnhold	: BOOL;
	(* This should be set to true if an external source requests that the module
	exit its current state and come to a controlled stop. Once set to true, the
	state machine will move to the 'Stopping' state. *)
	bStop	: BOOL;
	(* This should be set to true if a potentially hazardous error or a safety
	fault has occurred in any tasks. Once set to true, the state machine will
	move to the 'Aborting' state. *)
	bAbort	: BOOL;
END_VAR
// Unhold if the start button is pressed
bUnhold := in_bStartBtn;

// Stop if the stop button is pressed
bStop := in_bStopBtn;

// If the device has an error, abort
IF ref_fbDevice.P_bError THEN
	THIS^.M_SetError(200, 'Error on fbDevice!');
	bAbort := TRUE;
	
// Abort if abort button is pressed
ELSIF in_bAbortBtn THEN
	THIS^.M_SetError(100, 'Abort button pressed!');
	bAbort := TRUE;
END_IF
END_METHOD

(* Runs for a single cycle when exiting the held state. *)
METHOD M412_Held_Exit : BOOL
END_METHOD

(* Runs for a single cycle when entering the unholding state. *)
METHOD M420_Unholding_Entry : BOOL
THIS^.M_LogMessage('Unholding');

// Reset device status variables
bDeviceProgramStarted := FALSE;
END_METHOD

(* In this state, the module and its components should be returned to the
scenario it was in before it entered the 'Holding' step so that the
'Execute' state can pick up where it left off. *)
METHOD M421_Unholding : BOOL
VAR_OUTPUT
	(* This should be set to true once the module is ready to restart
	execution. Once set to true, the state machine will move to the 'Execute'
	state. *)
	bUnheld	: BOOL;
	(* This should be set to true if an external source requests that the module
	exit its current state and come to a controlled stop. Once set to true, the
	state machine will move to the 'Stopping' state. *)
	bStop	: BOOL;
	(* This should be set to true if a potentially hazardous error or a safety
	fault has occurred in any tasks. Once set to true, the state machine will
	move to the 'Aborting' state. *)
	bAbort	: BOOL;
END_VAR
// Restart the device program
IF NOT bDeviceProgramStarted THEN
	bDeviceProgramStarted := ref_fbDevice.M_StartProgram();

// Once the program is started, unholding is finished
ELSE
	bUnheld := TRUE;
END_IF

// Stop if the stop button is pressed
bStop := in_bStopBtn;

// If the device has an error, abort
IF ref_fbDevice.P_bError THEN
	THIS^.M_SetError(200, 'Error on fbDevice!');
	bAbort := TRUE;
	
// Abort if abort button is pressed
ELSIF in_bAbortBtn THEN
	THIS^.M_SetError(100, 'Abort button pressed!');
	bAbort := TRUE;
END_IF
END_METHOD

(* Runs for a single cycle when exiting the unholding state. *)
METHOD M422_Unholding_Exit : BOOL
END_METHOD

(* Runs for a single cycle when entering the suspending state. *)
METHOD M500_Suspending_Entry : BOOL
THIS^.M_LogMessage('Suspending');

// Reset device state variables
bDeviceProgramPaused := FALSE;
END_METHOD

(* This state should safely pause task executions without completely ending or
resetting them. *)
METHOD M501_Suspending : BOOL
VAR_OUTPUT
	(* This should be set to true once all execution tasks are safely paused.
	Once set to true, the state machine will move to the 'Suspended' state. *)
	bSuspended	: BOOL;
	(* This should be set to true if an external source requests that the module
	exit its current state and come to a controlled stop. Once set to true, the
	state machine will move to the 'Stopping' state. *)
	bStop	: BOOL;
	(* This should be set to true if a potentially hazardous error or a safety
	fault has occurred in any tasks. Once set to true, the state machine will
	move to the 'Aborting' state. *)
	bAbort	: BOOL;
END_VAR
// Pause the device
IF NOT bDeviceProgramPaused THEN
	bDeviceProgramPaused := ref_fbDevice.M_PauseProgram();
	
// Once the device is paused, done suspending
ELSE
	bSuspended := TRUE;
END_IF

// Stop if the stop button is pressed
bStop := in_bStopBtn;

// If the device has an error, abort
IF ref_fbDevice.P_bError THEN
	THIS^.M_SetError(200, 'Error on fbDevice!');
	bAbort := TRUE;
	
// Abort if abort button is pressed
ELSIF in_bAbortBtn THEN
	THIS^.M_SetError(100, 'Abort button pressed!');
	bAbort := TRUE;
END_IF
END_METHOD

(* Runs for a single cycle when exiting the suspending state. *)
METHOD M502_Suspending_Exit : BOOL
END_METHOD

(* Runs for a single cycle when entering the suspended state. *)
METHOD M510_Suspended_Entry : BOOL
THIS^.M_LogMessage('Suspended');
END_METHOD

(* In this state the most recent execution status should be maintained while
awaiting an explicit 'Unsuspend' command once external conditions are satisfactory. *)
METHOD M511_Suspended : BOOL
VAR_OUTPUT
	(* This should be set to true if an explicit 'Unsuspend' command is received.
	Once set to true, the state machine will move to the 'Unsuspending' state. *)
	bUnsuspend	: BOOL;
	(* This should be set to true if an external source requests that the module
	exit its current state and come to a controlled stop. Once set to true, the
	state machine will move to the 'Stopping' state. *)
	bStop	: BOOL;
	(* This should be set to true if a potentially hazardous error or a safety
	fault has occurred in any tasks. Once set to true, the state machine will
	move to the 'Aborting' state. *)
	bAbort	: BOOL;
END_VAR
// Unsuspend if the start button is pressed
bUnsuspend := in_bStartBtn;

// Stop if the stop button is pressed
bStop := in_bStopBtn;

// If the device has an error, abort
IF ref_fbDevice.P_bError THEN
	THIS^.M_SetError(200, 'Error on fbDevice!');
	bAbort := TRUE;
	
// Abort if abort button is pressed
ELSIF in_bAbortBtn THEN
	THIS^.M_SetError(100, 'Abort button pressed!');
	bAbort := TRUE;
END_IF
END_METHOD

(* Runs for a single cycle when exiting the suspended state. *)
METHOD M512_Suspended_Exit : BOOL
END_METHOD

(* Runs for a single cycle when entering the unsuspending state. *)
METHOD M520_Unsuspending_Entry : BOOL
THIS^.M_LogMessage('Unsuspending');

// Reset device status variables
bDeviceProgramStarted := FALSE;
END_METHOD

(* In this state, the module and its components should be returned to the
scenario it was in before it entered the 'Suspending' step so that the
'Execute' state can pick up where it left off. *)
METHOD M521_Unsuspending : BOOL
VAR_OUTPUT
	(* This should be set to true once the module is ready to restart
	execution. Once set to true, the state machine will move to the 'Execute'
	state. *)
	bUnsuspended	: BOOL;
	(* This should be set to true if an external source requests that the module
	exit its current state and come to a controlled stop. Once set to true, the
	state machine will move to the 'Stopping' state. *)
	bStop	: BOOL;
	(* This should be set to true if a potentially hazardous error or a safety
	fault has occurred in any tasks. Once set to true, the state machine will
	move to the 'Aborting' state. *)
	bAbort	: BOOL;
END_VAR
// Restart the device program
IF NOT bDeviceProgramStarted THEN
	bDeviceProgramStarted := ref_fbDevice.M_StartProgram();

// Once the program is started, unsuspending is finished
ELSE
	bUnsuspended := TRUE;
END_IF

// Stop if the stop button is pressed
bStop := in_bStopBtn;

// If the device has an error, abort
IF ref_fbDevice.P_bError THEN
	THIS^.M_SetError(200, 'Error on fbDevice!');
	bAbort := TRUE;
	
// Abort if abort button is pressed
ELSIF in_bAbortBtn THEN
	THIS^.M_SetError(100, 'Abort button pressed!');
	bAbort := TRUE;
END_IF
END_METHOD

(* Runs for a single cycle when exiting the unsuspending state. *)
METHOD M522_Unsuspending_Exit : BOOL
END_METHOD

ACTION A_DeviceTestTracking:
// Check device error state
fbDeviceAborted(CLK:=ref_fbDevice.P_bError);
fbDeviceReset(CLK:=ref_fbDevice.P_bError);

// Check device connection state
fbDeviceConnected(CLK:=ref_fbDevice.P_bConnected);
fbDeviceDisconnected(CLK:=ref_fbDevice.P_bConnected);

// Check device enable state
fbDeviceEnabled(CLK:=ref_fbDevice.P_bEnabled);
fbDeviceDisabled(CLK:=ref_fbDevice.P_bEnabled);

// Check device power state
fbDevicePoweredOn(CLK:=ref_fbDevice.P_bPoweredOn);
fbDevicePoweredOff(CLK:=ref_fbDevice.P_bPoweredOn);

// Check device program load state
fbDeviceProgramLoaded(CLK:=(
	ref_fbDevice.P_strCurrentProgram = in_strProgram
	AND LEN(in_strProgram) > 0));
	
// Set outputs based on triggers
IF fbDeviceAborted.Q		THEN out_bAbortTested 		:= TRUE; END_IF
IF fbDeviceReset.Q			THEN out_bResetTested 		:= TRUE; END_IF
IF fbDeviceConnected.Q		THEN out_bConnectTested 	:= TRUE; END_IF
IF fbDeviceDisconnected.Q	THEN out_bDisconnectTested	:= TRUE; END_IF
IF fbDeviceEnabled.Q		THEN out_bEnableTested 		:= TRUE; END_IF
IF fbDeviceDisabled.Q		THEN out_bDisableTested 	:= TRUE; END_IF
IF fbDevicePoweredOn.Q		THEN out_bPowerOnTested 	:= TRUE; END_IF
IF fbDevicePoweredOff.Q		THEN out_bPowerOffTested 	:= TRUE; END_IF
IF fbDeviceProgramLoaded.Q	THEN out_bLoadProgramTested	:= TRUE; END_IF

// Set program control state outputs
IF enumLastState = E_ProgramState.Stopped THEN
	IF ref_fbDevice.P_enumProgramState = E_ProgramState.Running THEN
		out_bStartProgramTested := TRUE;
	END_IF
ELSIF enumLastState = E_ProgramState.Running THEN
	IF ref_fbDevice.P_enumProgramState = E_ProgramState.Stopped THEN
		out_bStopProgramTested := TRUE;
	ELSIF ref_fbDevice.P_enumProgramState = E_ProgramState.Paused THEN
		out_bPauseProgramTested := TRUE;
	END_IF
ELSIF enumLastState = E_ProgramState.Paused THEN
	IF ref_fbDevice.P_enumProgramState = E_ProgramState.Running THEN
		out_bUnpauseProgramTested := TRUE;
	ELSIF ref_fbDevice.P_enumProgramState = E_ProgramState.Stopped THEN
		out_bStopPausedProgramTested := TRUE;
	END_IF
END_IF
enumLastState := ref_fbDevice.P_enumProgramState;
END_ACTION

END_FUNCTION_BLOCK

// Concrete/FB_DeviceTestStation
FUNCTION_BLOCK FB_DeviceTestStation EXTENDS FB_SimpleStation
VAR_INPUT
	ref_fbDevice: REFERENCE TO FB_Device; // The device to be tested

	in_strProgram: T_MaxString; // Program to load when testing program loading
END_VAR
VAR_OUTPUT
	out_bAbortTested: BOOL; // Gets set to TRUE once M_Abort on ref_fbDevice has been tested once
	
	out_bConnectTested: BOOL;  // Gets set to TRUE once M_Connect on ref_fbDevice has been tested once
	out_bDisconnectTested: BOOL;  // Gets set to TRUE once M_Disconnect on ref_fbDevice has been tested once
	
	out_bEnableTested: BOOL; // Gets set to TRUE once M_Enable on ref_fbDevice has been tested once
	out_bDisableTested: BOOL; // Gets set to TRUE once M_Disable on ref_fbDevice has been tested once
	
	out_bPowerOnTested: BOOL; // Gets set to TRUE once M_PowerOn on ref_fbDevice has been tested once
	out_bPowerOffTested: BOOL; // Gets set to TRUE once M_PowerOff on ref_fbDevice has been tested once
	
	out_bLoadProgramTested: BOOL; // Gets set to TRUE once M_LoadProgram on ref_fbDevice has been tested once
	out_bStartProgramTested: BOOL; // Gets set to TRUE once M_StartProgram on ref_fbDevice has been tested once
	out_bStopProgramTested: BOOL; // Gets set to TRUE once M_StopProgram on ref_fbDevice has been tested once
	out_bPauseProgramTested: BOOL; // Gets set to TRUE once M_PauseProgram on ref_fbDevice has been tested once
	out_bUnpauseProgramTested: BOOL; // Gets set to TRUE once M_StartProgram on ref_fbDevice has been tested once after M_PauseProgram was used
	out_bStopPausedProgramTested: BOOL; // Gets set to TRUE once M_StopProgram on ref_fbDevice has been tested once after M_PauseProgram was used
	
	out_bResetTested: BOOL; // Gets set to TRUE once M_Reset on ref_fbDevice has been tested once
END_VAR
VAR
	bDeviceReset: BOOL;
	
	bDeviceConnected: BOOL;
	bDeviceDisconnected: BOOL;
	
	bDevicePoweredOn: BOOL;
	bDevicePoweredOff: BOOL;
	
	bDeviceEnabled: BOOL;
	bDeviceDisabled: BOOL;
	
	bDeviceProgramLoaded: BOOL;
	bDeviceProgramStarted: BOOL;
	bDeviceProgramStopped: BOOL;
	bDeviceProgramPaused: BOOL;

	// Device test trackers
	fbDeviceAborted: R_TRIG;
	fbDeviceReset: F_TRIG;
	fbDeviceConnected: R_TRIG;
	fbDeviceDisconnected: F_TRIG;
	fbDeviceEnabled: R_TRIG;
	fbDeviceDisabled: F_TRIG;
	fbDevicePoweredOn: R_TRIG;
	fbDevicePoweredOff: F_TRIG;
	fbDeviceProgramLoaded: R_TRIG;
	enumLastState: E_ProgramState;
END_VAR

THIS^.M_SetDevice(1, ref_fbDevice);
THIS^.M_SetInitialDeviceProgram(1, in_strProgram);

A_RunSimpleStation();

A_DeviceTestTracking();

ACTION A_DeviceTestTracking:
// Check device error state
fbDeviceAborted(CLK:=ref_fbDevice.P_bError);
fbDeviceReset(CLK:=ref_fbDevice.P_bError);

// Check device connection state
fbDeviceConnected(CLK:=ref_fbDevice.P_bConnected);
fbDeviceDisconnected(CLK:=ref_fbDevice.P_bConnected);

// Check device enable state
fbDeviceEnabled(CLK:=ref_fbDevice.P_bEnabled);
fbDeviceDisabled(CLK:=ref_fbDevice.P_bEnabled);

// Check device power state
fbDevicePoweredOn(CLK:=ref_fbDevice.P_bPoweredOn);
fbDevicePoweredOff(CLK:=ref_fbDevice.P_bPoweredOn);

// Check device program load state
fbDeviceProgramLoaded(CLK:=(
	ref_fbDevice.P_strCurrentProgram = in_strProgram
	AND LEN(in_strProgram) > 0));
	
// Set outputs based on triggers
IF fbDeviceAborted.Q		THEN out_bAbortTested 		:= TRUE; END_IF
IF fbDeviceReset.Q			THEN out_bResetTested 		:= TRUE; END_IF
IF fbDeviceConnected.Q		THEN out_bConnectTested 	:= TRUE; END_IF
IF fbDeviceDisconnected.Q	THEN out_bDisconnectTested	:= TRUE; END_IF
IF fbDeviceEnabled.Q		THEN out_bEnableTested 		:= TRUE; END_IF
IF fbDeviceDisabled.Q		THEN out_bDisableTested 	:= TRUE; END_IF
IF fbDevicePoweredOn.Q		THEN out_bPowerOnTested 	:= TRUE; END_IF
IF fbDevicePoweredOff.Q		THEN out_bPowerOffTested 	:= TRUE; END_IF
IF fbDeviceProgramLoaded.Q	THEN out_bLoadProgramTested	:= TRUE; END_IF

// Set program control state outputs
IF enumLastState = E_ProgramState.Stopped THEN
	IF ref_fbDevice.P_enumProgramState = E_ProgramState.Running THEN
		out_bStartProgramTested := TRUE;
	END_IF
ELSIF enumLastState = E_ProgramState.Running THEN
	IF ref_fbDevice.P_enumProgramState = E_ProgramState.Stopped THEN
		out_bStopProgramTested := TRUE;
	ELSIF ref_fbDevice.P_enumProgramState = E_ProgramState.Paused THEN
		out_bPauseProgramTested := TRUE;
	END_IF
ELSIF enumLastState = E_ProgramState.Paused THEN
	IF ref_fbDevice.P_enumProgramState = E_ProgramState.Running THEN
		out_bUnpauseProgramTested := TRUE;
	ELSIF ref_fbDevice.P_enumProgramState = E_ProgramState.Stopped THEN
		out_bStopPausedProgramTested := TRUE;
	END_IF
END_IF
enumLastState := ref_fbDevice.P_enumProgramState;
END_ACTION

END_FUNCTION_BLOCK

// Concrete/FB_SimpleStation
(*
	Simple station that extends adds buttons to FB_Machine
*)
{attribute 'hide_all_locals'}
FUNCTION_BLOCK FB_SimpleStation EXTENDS FB_Station
VAR_INPUT
	(* Immediately abort all stations from whatever state they are in and
		go to the Aborted state. *)
	in_bAbortBtn : BOOL;
	(* Immediately stop all stations from whatever state they are in and
		go to the Stopped state. *)
	in_bStopBtn : BOOL;
	(* Clear all stations from the Aborted state and go to the Stopped state. *)
	in_bClearBtn : BOOL;
	(* Reset all stations from the Stopped state and go to the Idle state. *)
	in_bResetBtn : BOOL;
	(* Start all stations from the Idle state and go to the Execute state. *)
	in_bStartBtn : BOOL;
	(* Hold all stations from the Execute state and go to the Held state. *)
	in_bHoldBtn : BOOL;
	(* Unhold all stations from the Held state and go to the Execute state. *)
	in_bUnholdBtn : BOOL;
	(* Suspend all stations from the Execute state and go to the Held Suspended. *)
	in_bSuspendBtn : BOOL;
	(* Unsuspend all stations from the Suspended state and go to the Execute state. *)
	in_bUnsuspendBtn : BOOL;
	(* Complete all stations from the Execute state and go to the Completed state. *)
	in_bCompleteBtn : BOOL;
	(* Return all stations from the Completed state and go to the Idle state. *)
	in_bReturnBtn : BOOL;
END_VAR
VAR_OUTPUT
END_VAR
VAR
	// Abort
	ssta_fbAbortTrig: R_TRIG;
	ssta_bAbortTrig: BOOL;
	ssta_bAborting: BOOL;
	ssta_bAborted: BOOL;

	// Stop
	ssta_fbStopTrig: R_TRIG;
	ssta_bStopTrig: BOOL;
	ssta_bStopping: BOOL;
	ssta_bStopped: BOOL;
	
	// Aborted
	ssta_fbClearTrig: R_TRIG;
	ssta_bClearTrig: BOOL;
	
	// Stopped
	ssta_fbResetTrig: R_TRIG;
	ssta_bResetTrig: BOOL;
	
	// Idle
	ssta_fbStartTrig: R_TRIG;
	ssta_bStartTrig: BOOL;
	
	// Execute
	ssta_fbCompleteTrig: R_TRIG;
	ssta_bCompleteTrig: BOOL;
	ssta_fbHoldTrig: R_TRIG;
	ssta_bHoldTrig: BOOL;
	ssta_fbSuspendTrig: R_TRIG;
	ssta_bSuspendTrig: BOOL;
	
	// Complete
	ssta_fbReturnTrig: R_TRIG;
	ssta_bReturnTrig: BOOL;
	
	// Held
	ssta_fbUnholdTrig: R_TRIG;
	ssta_bUnholdTrig: BOOL;
	
	// Suspended
	ssta_fbUnsuspendTrig: R_TRIG;
	ssta_bUnsuspendTrig: BOOL;
END_VAR

THIS^.A_RunSimpleStation();

ACTION A_Buttons:
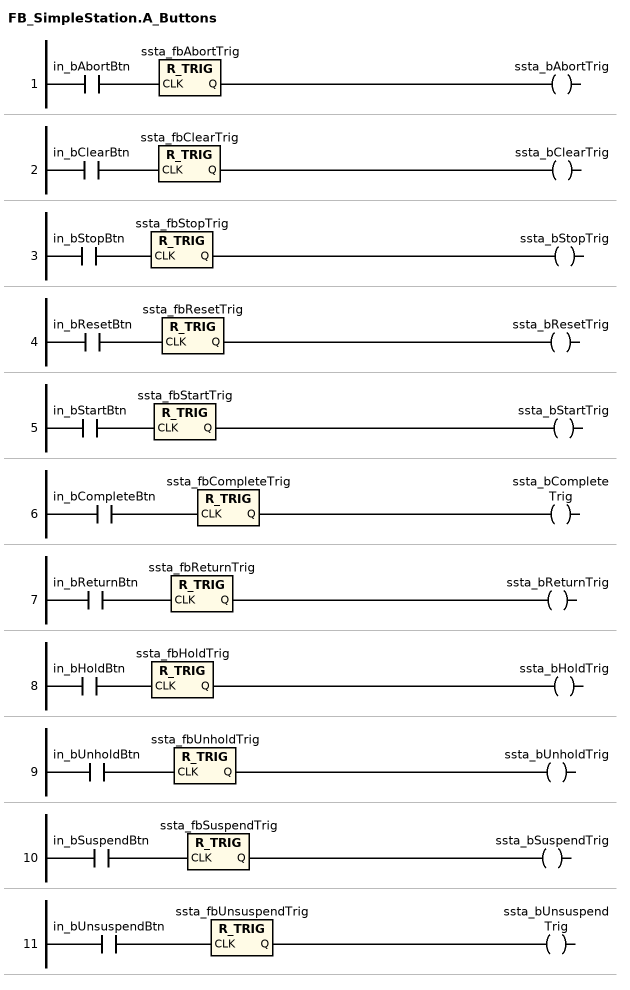
// NETWORK 1
ssta_fbAbortTrig(CLK := in_bAbortBtn); // R_TRIG
ssta_bAbortTrig := ssta_fbAbortTrig.Q;

// NETWORK 2
ssta_fbClearTrig(CLK := in_bClearBtn); // R_TRIG
ssta_bClearTrig := ssta_fbClearTrig.Q;

// NETWORK 3
ssta_fbStopTrig(CLK := in_bStopBtn); // R_TRIG
ssta_bStopTrig := ssta_fbStopTrig.Q;

// NETWORK 4
ssta_fbResetTrig(CLK := in_bResetBtn); // R_TRIG
ssta_bResetTrig := ssta_fbResetTrig.Q;

// NETWORK 5
ssta_fbStartTrig(CLK := in_bStartBtn); // R_TRIG
ssta_bStartTrig := ssta_fbStartTrig.Q;

// NETWORK 6
ssta_fbCompleteTrig(CLK := in_bCompleteBtn); // R_TRIG
ssta_bCompleteTrig := ssta_fbCompleteTrig.Q;

// NETWORK 7
ssta_fbReturnTrig(CLK := in_bReturnBtn); // R_TRIG
ssta_bReturnTrig := ssta_fbReturnTrig.Q;

// NETWORK 8
ssta_fbHoldTrig(CLK := in_bHoldBtn); // R_TRIG
ssta_bHoldTrig := ssta_fbHoldTrig.Q;

// NETWORK 9
ssta_fbUnholdTrig(CLK := in_bUnholdBtn); // R_TRIG
ssta_bUnholdTrig := ssta_fbUnholdTrig.Q;

// NETWORK 10
ssta_fbSuspendTrig(CLK := in_bSuspendBtn); // R_TRIG
ssta_bSuspendTrig := ssta_fbSuspendTrig.Q;

// NETWORK 11
ssta_fbUnsuspendTrig(CLK := in_bUnsuspendBtn); // R_TRIG
ssta_bUnsuspendTrig := ssta_fbUnsuspendTrig.Q;
END_ACTION

ACTION A_RunSimpleStation:
THIS^.A_StopAndAbort();
THIS^.A_Buttons();
THIS^.A_StateMachine();
END_ACTION

ACTION A_StopAndAbort:
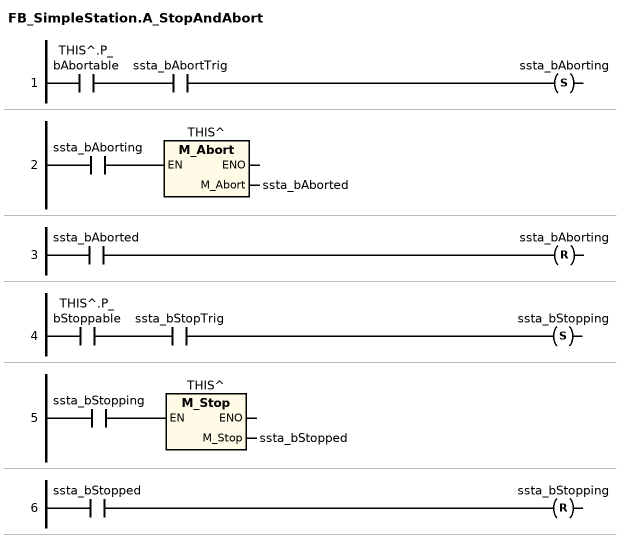
// NETWORK 1
ssta_bAborting S= THIS^.P_bAbortable AND ssta_bAbortTrig;

// NETWORK 2
IF ssta_bAborting THEN THIS^.M_Abort(M_Abort => ssta_bAborted); END_IF

// NETWORK 3
ssta_bAborting R= ssta_bAborted;

// NETWORK 4
ssta_bStopping S= THIS^.P_bStoppable AND ssta_bStopTrig;

// NETWORK 5
IF ssta_bStopping THEN THIS^.M_Stop(M_Stop => ssta_bStopped); END_IF

// NETWORK 6
ssta_bStopping R= ssta_bStopped;
END_ACTION

(* This state is entered after the aborting state completes, and should
not modify anything in the module while awaiting an explicit 'Clear' command. *)
METHOD M011_Aborted : BOOL
VAR_OUTPUT
	(* This should be set to true once an explicit 'Clear' command is received.
	Once set to true, the state machine will move to the 'Clearing' state. *)
	bClear	: BOOL;
END_VAR
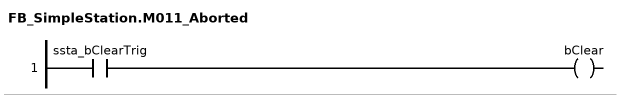
// NETWORK 1
bClear := ssta_bClearTrig;
END_METHOD

(* The machine should be stationary and awaiting an explicit 'Reset' command
while in this state. Once the 'Reset' command is received, the state machine
will move to the 'Resetting' state. *)
METHOD M111_Stopped : BOOL
VAR_OUTPUT
	(* This should be set to true if an explicit reset command is received.
	Once set to true, the state machine will move to the 'Resetting' state. *)
	bReset	: BOOL;
	(* This should be set to true if a potentially hazardous error or a safety
	fault has occurred in any tasks. Once set to true, the state machine will
	move to the 'Aborting' state. *)
	bAbort	: BOOL;
END_VAR
VAR
	_bDeviceError: BOOL;
	_strDeviceErrorId: T_MaxString;
	_udintDeviceErrorCode: UDINT;
	_strDeviceErrorMsg: T_MaxString;
	_strErrorMsg: STRING(255);
END_VAR
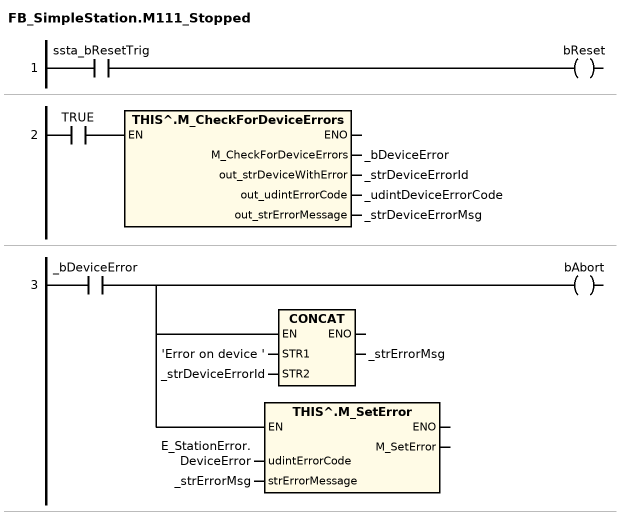
// NETWORK 1
bReset := ssta_bResetTrig;

// NETWORK 2
_bDeviceError := THIS^.M_CheckForDeviceErrors(out_strDeviceWithError => _strDeviceErrorId, out_udintErrorCode => _udintDeviceErrorCode, out_strErrorMessage => _strDeviceErrorMsg);

// NETWORK 3
bAbort := _bDeviceError;
IF _bDeviceError THEN _strErrorMsg := CONCAT(STR1 := 'Error on device ', STR2 := _strDeviceErrorId); END_IF
IF _bDeviceError THEN
    THIS^.M_SetError(udintErrorCode := E_StationError.DeviceError, strErrorMessage := _strErrorMsg);
END_IF
END_METHOD

(* This state should maintain the status of the module and its components that
was set by the resetting step while awaiting an explicit 'Start' command. *)
METHOD M211_Idle : BOOL
VAR_OUTPUT
	(* This should be set to true if an explicit 'Start' command is received.
	Once set to true, the state machine will move to the 'Starting' state. *)
	bStart	: BOOL;
	(* This should be set to true if an external source requests that the module
	exit its current state and come to a controlled stop. Once set to true, the
	state machine will move to the 'Stopping' state. *)
	bStop	: BOOL;
	(* This should be set to true if a potentially hazardous error or a safety
	fault has occurred in any tasks. Once set to true, the state machine will
	move to the 'Aborting' state. *)
	bAbort	: BOOL;
END_VAR
VAR
	_bDeviceError: BOOL;
	_strDeviceErrorId: T_MaxString;
	_udintDeviceErrorCode: UDINT;
	_strDeviceErrorMsg: T_MaxString;
	_strErrorMsg: STRING(255);
END_VAR
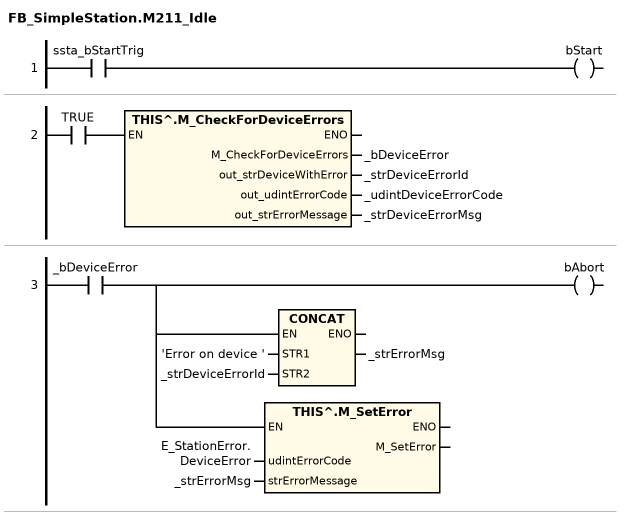
// NETWORK 1
bStart := ssta_bStartTrig;

// NETWORK 2
_bDeviceError := THIS^.M_CheckForDeviceErrors(out_strDeviceWithError => _strDeviceErrorId, out_udintErrorCode => _udintDeviceErrorCode, out_strErrorMessage => _strDeviceErrorMsg);

// NETWORK 3
bAbort := _bDeviceError;
IF _bDeviceError THEN _strErrorMsg := CONCAT(STR1 := 'Error on device ', STR2 := _strDeviceErrorId); END_IF
IF _bDeviceError THEN
    THIS^.M_SetError(udintErrorCode := E_StationError.DeviceError, strErrorMessage := _strErrorMsg);
END_IF
END_METHOD

(* The module should remain in this state while it is actively performing
automated tasks. Once all work is finished the state machine should move to the
'Completing' state. *)
METHOD M311_Execute : BOOL
VAR_OUTPUT
	(* This should be set to true once all tasks are complete and automated
	execution should be ended. Once set to true, the state machine will move to
	the 'Completing' state. *)
	bFinished	: BOOL;
	(* This should be set to true as a result of an explicit 'Hold' command
	or if internal conditions require the module to stop operation without
	completely exiting the execution sequence. Once set to true, the state
	machine will move to the 'Holding' state. *)
	bHold	: BOOL;
	(* This should be set to true if external conditions require the module to
	suspend operation until the external conditions are cleared. Once set to
	true, the state machine will move to the 'Suspending' state. *)
	bSuspend	: BOOL;
	(* This should be set to true if an external source requests that the module
	exit its current state and come to a controlled stop. Once set to true, the
	state machine will move to the 'Stopping' state. *)
	bStop	: BOOL;
	(* This should be set to true if a potentially hazardous error or a safety
	fault has occurred in any tasks. Once set to true, the state machine will
	move to the 'Aborting' state. *)
	bAbort	: BOOL;
END_VAR
VAR
	_bDeviceError: BOOL;
	_strDeviceErrorId: T_MaxString;
	_udintDeviceErrorCode: UDINT;
	_strDeviceErrorMsg: T_MaxString;
	_strErrorMsg: STRING(255);
END_VAR
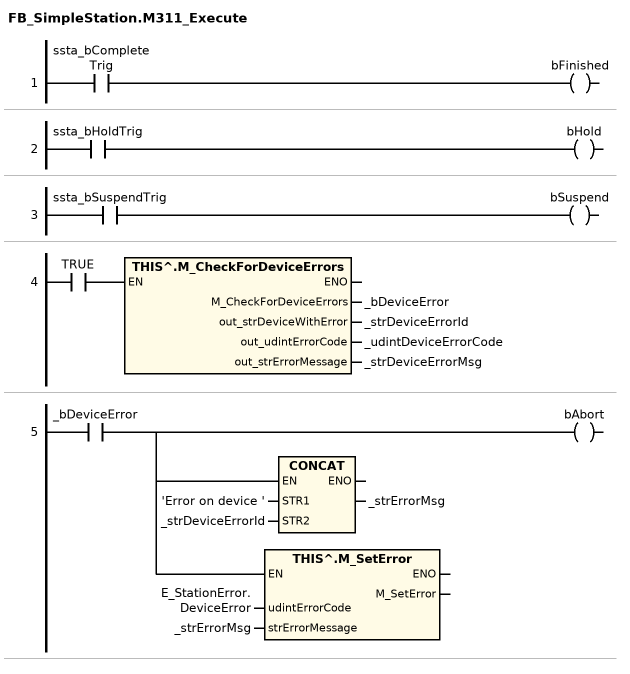
// NETWORK 1
bFinished := ssta_bCompleteTrig;

// NETWORK 2
bHold := ssta_bHoldTrig;

// NETWORK 3
bSuspend := ssta_bSuspendTrig;

// NETWORK 4
_bDeviceError := THIS^.M_CheckForDeviceErrors(out_strDeviceWithError => _strDeviceErrorId, out_udintErrorCode => _udintDeviceErrorCode, out_strErrorMessage => _strDeviceErrorMsg);

// NETWORK 5
bAbort := _bDeviceError;
IF _bDeviceError THEN _strErrorMsg := CONCAT(STR1 := 'Error on device ', STR2 := _strDeviceErrorId); END_IF
IF _bDeviceError THEN
    THIS^.M_SetError(udintErrorCode := E_StationError.DeviceError, strErrorMessage := _strErrorMsg);
END_IF
END_METHOD

(* The module should remain stationary within this state while maintaing any
execution statistics and awaiting an explicit 'Return' command. *)
METHOD M331_Complete : BOOL
VAR_OUTPUT
	(* This should be set to true if an explicit 'Return' command is received.
	Once set to true, the state machine will move to the 'Resetting' state. *)
	bReturn	: BOOL;
	(* This should be set to true if an external source requests that the module
	exit its current state and come to a controlled stop. Once set to true, the
	state machine will move to the 'Stopping' state. *)
	bStop	: BOOL;
	(* This should be set to true if a potentially hazardous error or a safety
	fault has occurred in any tasks. Once set to true, the state machine will
	move to the 'Aborting' state. *)
	bAbort	: BOOL;
END_VAR
VAR
	_bDeviceError: BOOL;
	_strDeviceErrorId: T_MaxString;
	_udintDeviceErrorCode: UDINT;
	_strDeviceErrorMsg: T_MaxString;
	_strErrorMsg: STRING(255);
END_VAR
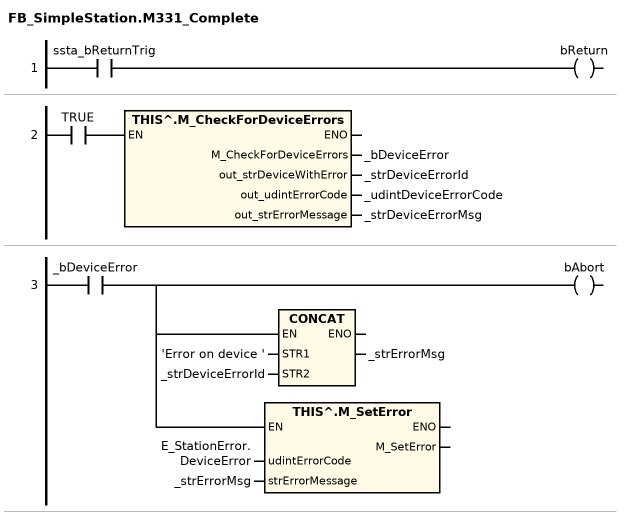
// NETWORK 1
bReturn := ssta_bReturnTrig;

// NETWORK 2
_bDeviceError := THIS^.M_CheckForDeviceErrors(out_strDeviceWithError => _strDeviceErrorId, out_udintErrorCode => _udintDeviceErrorCode, out_strErrorMessage => _strDeviceErrorMsg);

// NETWORK 3
bAbort := _bDeviceError;
IF _bDeviceError THEN _strErrorMsg := CONCAT(STR1 := 'Error on device ', STR2 := _strDeviceErrorId); END_IF
IF _bDeviceError THEN
    THIS^.M_SetError(udintErrorCode := E_StationError.DeviceError, strErrorMessage := _strErrorMsg);
END_IF
END_METHOD

(* In this state the most recent execution status should be maintained while
awaiting an explicit 'Unhold' command once internal conditions are satisfactory. *)
METHOD M411_Held : BOOL
VAR_OUTPUT
	(* This should be set to true if an explicit 'Unhold' command is received.
	Once set to true, the state machine will move to the 'Unholding' state. *)
	bUnhold	: BOOL;
	(* This should be set to true if an external source requests that the module
	exit its current state and come to a controlled stop. Once set to true, the
	state machine will move to the 'Stopping' state. *)
	bStop	: BOOL;
	(* This should be set to true if a potentially hazardous error or a safety
	fault has occurred in any tasks. Once set to true, the state machine will
	move to the 'Aborting' state. *)
	bAbort	: BOOL;
END_VAR
VAR
	_bDeviceError: BOOL;
	_strDeviceErrorId: T_MaxString;
	_udintDeviceErrorCode: UDINT;
	_strDeviceErrorMsg: T_MaxString;
	_strErrorMsg: STRING(255);
END_VAR
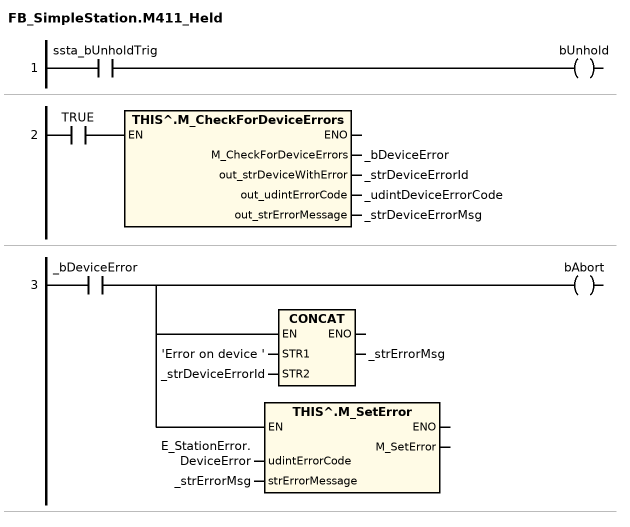
// NETWORK 1
bUnhold := ssta_bUnholdTrig;

// NETWORK 2
_bDeviceError := THIS^.M_CheckForDeviceErrors(out_strDeviceWithError => _strDeviceErrorId, out_udintErrorCode => _udintDeviceErrorCode, out_strErrorMessage => _strDeviceErrorMsg);

// NETWORK 3
bAbort := _bDeviceError;
IF _bDeviceError THEN _strErrorMsg := CONCAT(STR1 := 'Error on device ', STR2 := _strDeviceErrorId); END_IF
IF _bDeviceError THEN
    THIS^.M_SetError(udintErrorCode := E_StationError.DeviceError, strErrorMessage := _strErrorMsg);
END_IF
END_METHOD

(* In this state the most recent execution status should be maintained while
awaiting an explicit 'Unsuspend' command once external conditions are satisfactory. *)
METHOD M511_Suspended : BOOL
VAR_OUTPUT
	(* This should be set to true if an explicit 'Unsuspend' command is received.
	Once set to true, the state machine will move to the 'Unsuspending' state. *)
	bUnsuspend	: BOOL;
	(* This should be set to true if an external source requests that the module
	exit its current state and come to a controlled stop. Once set to true, the
	state machine will move to the 'Stopping' state. *)
	bStop	: BOOL;
	(* This should be set to true if a potentially hazardous error or a safety
	fault has occurred in any tasks. Once set to true, the state machine will
	move to the 'Aborting' state. *)
	bAbort	: BOOL;
END_VAR
VAR
	_bDeviceError: BOOL;
	_strDeviceErrorId: T_MaxString;
	_udintDeviceErrorCode: UDINT;
	_strDeviceErrorMsg: T_MaxString;
	_strErrorMsg: STRING(255);
END_VAR
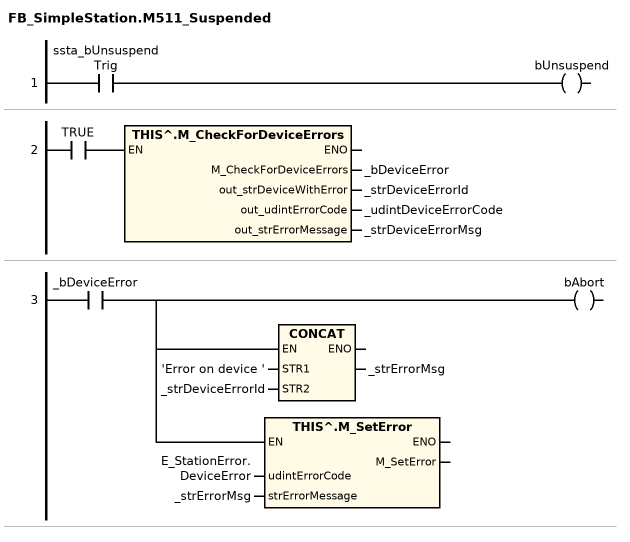
// NETWORK 1
bUnsuspend := ssta_bUnsuspendTrig;

// NETWORK 2
_bDeviceError := THIS^.M_CheckForDeviceErrors(out_strDeviceWithError => _strDeviceErrorId, out_udintErrorCode => _udintDeviceErrorCode, out_strErrorMessage => _strDeviceErrorMsg);

// NETWORK 3
bAbort := _bDeviceError;
IF _bDeviceError THEN _strErrorMsg := CONCAT(STR1 := 'Error on device ', STR2 := _strDeviceErrorId); END_IF
IF _bDeviceError THEN
    THIS^.M_SetError(udintErrorCode := E_StationError.DeviceError, strErrorMessage := _strErrorMsg);
END_IF
END_METHOD

END_FUNCTION_BLOCK

// Concrete/FB_SimpleMachine
(*
	Simple machine that extends adds buttons to FB_Machine
*)
{attribute 'hide_all_locals'}
FUNCTION_BLOCK FB_SimpleMachine EXTENDS FB_Machine IMPLEMENTS I_SimpleWaitingStatesOnly
VAR_INPUT
	(* Immediately abort all stations from whatever state they are in and
		go to the Aborted state. *)
	in_bAbortBtn : BOOL;
	(* Immediately stop all stations from whatever state they are in and
		go to the Stopped state. *)
	in_bStopBtn : BOOL;
	(* Clear all stations from the Aborted state and go to the Stopped state. *)
	in_bClearBtn : BOOL;
	(* Reset all stations from the Stopped state and go to the Idle state. *)
	in_bResetBtn : BOOL;
	(* Start all stations from the Idle state and go to the Execute state. *)
	in_bStartBtn : BOOL;
	(* Hold all stations from the Execute state and go to the Held state. *)
	in_bHoldBtn : BOOL;
	(* Unhold all stations from the Held state and go to the Execute state. *)
	in_bUnholdBtn : BOOL;
	(* Suspend all stations from the Execute state and go to the Held Suspended. *)
	in_bSuspendBtn : BOOL;
	(* Unsuspend all stations from the Suspended state and go to the Execute state. *)
	in_bUnsuspendBtn : BOOL;
	(* Complete all stations from the Execute state and go to the Completed state. *)
	in_bCompleteBtn : BOOL;
	(* Return all stations from the Completed state and go to the Idle state. *)
	in_bReturnBtn : BOOL;
END_VAR
VAR_OUTPUT
END_VAR
VAR
	// Abort
	smac_fbAbortTrig: R_TRIG;
	smac_bAbortTrig: BOOL;
	smac_bAborting: BOOL;
	smac_bAborted: BOOL;

	// Stop
	smac_fbStopTrig: R_TRIG;
	smac_bStopTrig: BOOL;
	smac_bStopping: BOOL;
	smac_bStopped: BOOL;
	
	// Aborted
	smac_fbClearTrig: R_TRIG;
	smac_bClearTrig: BOOL;
	
	// Stopped
	smac_fbResetTrig: R_TRIG;
	smac_bResetTrig: BOOL;
	
	// Idle
	smac_fbStartTrig: R_TRIG;
	smac_bStartTrig: BOOL;
	
	// Execute
	smac_fbCompleteTrig: R_TRIG;
	smac_bCompleteTrig: BOOL;
	smac_fbHoldTrig: R_TRIG;
	smac_bHoldTrig: BOOL;
	smac_fbSuspendTrig: R_TRIG;
	smac_bSuspendTrig: BOOL;
	
	// Complete
	smac_fbReturnTrig: R_TRIG;
	smac_bReturnTrig: BOOL;
	
	// Held
	smac_fbUnholdTrig: R_TRIG;
	smac_bUnholdTrig: BOOL;
	
	// Suspended
	smac_fbUnsuspendTrig: R_TRIG;
	smac_bUnsuspendTrig: BOOL;
END_VAR

THIS^.A_RunSimpleMachine();

ACTION A_Buttons:
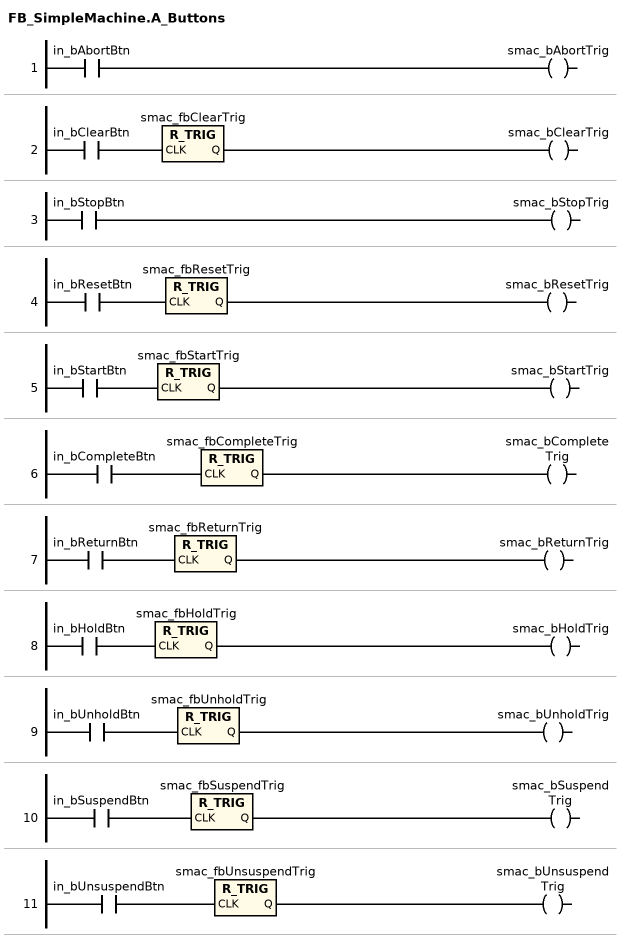
// NETWORK 1
smac_bAbortTrig := in_bAbortBtn;

// NETWORK 2
smac_fbClearTrig(CLK := in_bClearBtn); // R_TRIG
smac_bClearTrig := smac_fbClearTrig.Q;

// NETWORK 3
smac_bStopTrig := in_bStopBtn;

// NETWORK 4
smac_fbResetTrig(CLK := in_bResetBtn); // R_TRIG
smac_bResetTrig := smac_fbResetTrig.Q;

// NETWORK 5
smac_fbStartTrig(CLK := in_bStartBtn); // R_TRIG
smac_bStartTrig := smac_fbStartTrig.Q;

// NETWORK 6
smac_fbCompleteTrig(CLK := in_bCompleteBtn); // R_TRIG
smac_bCompleteTrig := smac_fbCompleteTrig.Q;

// NETWORK 7
smac_fbReturnTrig(CLK := in_bReturnBtn); // R_TRIG
smac_bReturnTrig := smac_fbReturnTrig.Q;

// NETWORK 8
smac_fbHoldTrig(CLK := in_bHoldBtn); // R_TRIG
smac_bHoldTrig := smac_fbHoldTrig.Q;

// NETWORK 9
smac_fbUnholdTrig(CLK := in_bUnholdBtn); // R_TRIG
smac_bUnholdTrig := smac_fbUnholdTrig.Q;

// NETWORK 10
smac_fbSuspendTrig(CLK := in_bSuspendBtn); // R_TRIG
smac_bSuspendTrig := smac_fbSuspendTrig.Q;

// NETWORK 11
smac_fbUnsuspendTrig(CLK := in_bUnsuspendBtn); // R_TRIG
smac_bUnsuspendTrig := smac_fbUnsuspendTrig.Q;
END_ACTION

ACTION A_RunSimpleMachine:
THIS^.A_StopAndAbort();
THIS^.A_Buttons();
THIS^.A_StateMachine();
END_ACTION

ACTION A_StopAndAbort:
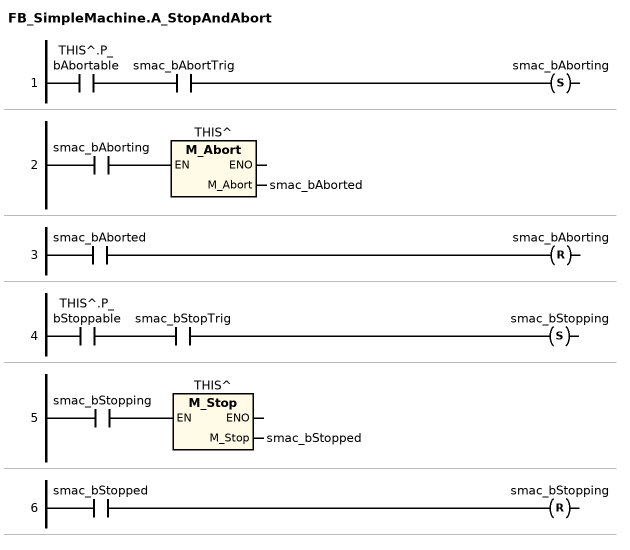
// NETWORK 1
smac_bAborting S= THIS^.P_bAbortable AND smac_bAbortTrig;

// NETWORK 2
IF smac_bAborting THEN THIS^.M_Abort(M_Abort => smac_bAborted); END_IF

// NETWORK 3
smac_bAborting R= smac_bAborted;

// NETWORK 4
smac_bStopping S= THIS^.P_bStoppable AND smac_bStopTrig;

// NETWORK 5
IF smac_bStopping THEN THIS^.M_Stop(M_Stop => smac_bStopped); END_IF

// NETWORK 6
smac_bStopping R= smac_bStopped;
END_ACTION

(* This state is entered after the aborting state completes, and should
not modify anything in the module while awaiting an explicit 'Clear' command. *)
METHOD M011_Aborted : BOOL
VAR_OUTPUT
	(* This should be set to true once an explicit 'Clear' command is received.
	Once set to true, the state machine will move to the 'Clearing' state. *)
	bClear	: BOOL;
END_VAR
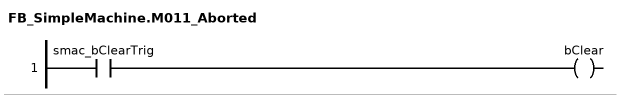
// NETWORK 1
bClear := smac_bClearTrig;
END_METHOD

(* The machine should be stationary and awaiting an explicit 'Reset' command
while in this state. Once the 'Reset' command is received, the state machine
will move to the 'Resetting' state. *)
METHOD M111_Stopped : BOOL
VAR_OUTPUT
	(* This should be set to true if an explicit reset command is received.
	Once set to true, the state machine will move to the 'Resetting' state. *)
	bReset	: BOOL;
	(* This should be set to true if a potentially hazardous error or a safety
	fault has occurred in any tasks. Once set to true, the state machine will
	move to the 'Aborting' state. *)
	bAbort	: BOOL;
END_VAR
VAR
	_bStationError: BOOL;
END_VAR
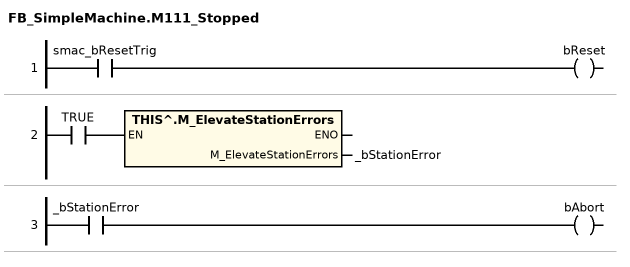
// NETWORK 1
bReset := smac_bResetTrig;

// NETWORK 2
_bStationError := THIS^.M_ElevateStationErrors();

// NETWORK 3
bAbort := _bStationError;
END_METHOD

(* This state should maintain the status of the module and its components that
was set by the resetting step while awaiting an explicit 'Start' command. *)
METHOD M211_Idle : BOOL
VAR_OUTPUT
	(* This should be set to true if an explicit 'Start' command is received.
	Once set to true, the state machine will move to the 'Starting' state. *)
	bStart	: BOOL;
	(* This should be set to true if an external source requests that the module
	exit its current state and come to a controlled stop. Once set to true, the
	state machine will move to the 'Stopping' state. *)
	bStop	: BOOL;
	(* This should be set to true if a potentially hazardous error or a safety
	fault has occurred in any tasks. Once set to true, the state machine will
	move to the 'Aborting' state. *)
	bAbort	: BOOL;
END_VAR
VAR
	_bStationError: BOOL;
END_VAR
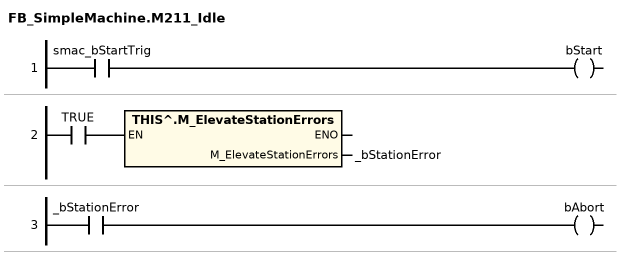
// NETWORK 1
bStart := smac_bStartTrig;

// NETWORK 2
_bStationError := THIS^.M_ElevateStationErrors();

// NETWORK 3
bAbort := _bStationError;
END_METHOD

(* The module should remain in this state while it is actively performing
automated tasks. Once all work is finished the state machine should move to the
'Completing' state. *)
METHOD M311_Execute : BOOL
VAR_OUTPUT
	(* This should be set to true once all tasks are complete and automated
	execution should be ended. Once set to true, the state machine will move to
	the 'Completing' state. *)
	bFinished	: BOOL;
	(* This should be set to true as a result of an explicit 'Hold' command
	or if internal conditions require the module to stop operation without
	completely exiting the execution sequence. Once set to true, the state
	machine will move to the 'Holding' state. *)
	bHold	: BOOL;
	(* This should be set to true if external conditions require the module to
	suspend operation until the external conditions are cleared. Once set to
	true, the state machine will move to the 'Suspending' state. *)
	bSuspend	: BOOL;
	(* This should be set to true if an external source requests that the module
	exit its current state and come to a controlled stop. Once set to true, the
	state machine will move to the 'Stopping' state. *)
	bStop	: BOOL;
	(* This should be set to true if a potentially hazardous error or a safety
	fault has occurred in any tasks. Once set to true, the state machine will
	move to the 'Aborting' state. *)
	bAbort	: BOOL;
END_VAR
VAR
	_bStationError: BOOL;
END_VAR
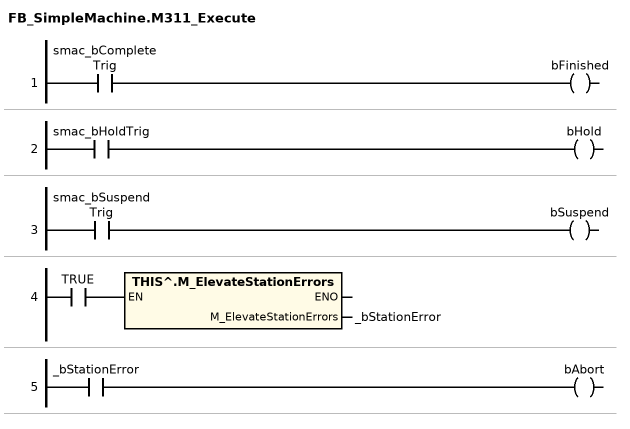
// NETWORK 1
bFinished := smac_bCompleteTrig;

// NETWORK 2
bHold := smac_bHoldTrig;

// NETWORK 3
bSuspend := smac_bSuspendTrig;

// NETWORK 4
_bStationError := THIS^.M_ElevateStationErrors();

// NETWORK 5
bAbort := _bStationError;
END_METHOD

(* The module should remain stationary within this state while maintaing any
execution statistics and awaiting an explicit 'Return' command. *)
METHOD M331_Complete : BOOL
VAR_OUTPUT
	(* This should be set to true if an explicit 'Return' command is received.
	Once set to true, the state machine will move to the 'Resetting' state. *)
	bReturn	: BOOL;
	(* This should be set to true if an external source requests that the module
	exit its current state and come to a controlled stop. Once set to true, the
	state machine will move to the 'Stopping' state. *)
	bStop	: BOOL;
	(* This should be set to true if a potentially hazardous error or a safety
	fault has occurred in any tasks. Once set to true, the state machine will
	move to the 'Aborting' state. *)
	bAbort	: BOOL;
END_VAR
VAR
	_bStationError: BOOL;
END_VAR
